(* Logix 5000 project; controller QW361 vendor 1 type 14 code 107 rev 32.11; software revision 32.00; part 9 of 20 *)

        [1052].log_data[0].time := 300.0, [1052].log_data[0].minminute := 10, [1052].log_data[0].maxminute := 10, [1052].log_data[0].valid := 1, [1052].log_data[1].valid := 1, [1052].log_data[2].valid := 1, [1052].log_data[3].valid := 1, [1052].log_data[4].valid := 1, [1052].time.Year := 2022, [1052].time.Month := 4, [1052].time.Day := 27, [1052].time.Hour := 13, [1052].time.Minute := 14, [1052].time.Second := 59, [1052].time.DST_ON := 1, [1053].log_data[0].min := 1.0, [1053].log_data[0].max := 1.0, [1053].log_data[0].total := 300.0, [1053].log_data[0].time := 300.0, [1053].log_data[0].minminute := 15, [1053].log_data[0].maxminute := 15, [1053].log_data[0].valid := 1, [1053].log_data[1].valid := 1, [1053].log_data[2].valid := 1, [1053].log_data[3].valid := 1, [1053].log_data[4].valid := 1, [1053].time.Year := 2022, [1053].time.Month := 4, [1053].time.Day := 27, [1053].time.Hour := 13, [1053].time.Minute := 19, [1053].time.Second := 59, [1053].time.DST_ON := 1, [1054].log_data[0].min := 1.0, [1054].log_data[0].max := 1.0, [1054].log_data[0].total := 300.0, [1054].log_data[0].time := 300.0, [1054].log_data[0].minminute := 20, [1054].log_data[0].maxminute := 20, [1054].log_data[0].valid := 1, [1054].log_data[1].valid := 1, [1054].log_data[2].valid := 1, [1054].log_data[3].valid := 1, [1054].log_data[4].valid := 1, [1054].time.Year := 2022, [1054].time.Month := 4, [1054].time.Day := 27, [1054].time.Hour := 13, [1054].time.Minute := 24, [1054].time.Second := 59, [1054].time.DST_ON := 1, [1055].log_data[0].min := 1.0, [1055].log_data[0].max := 1.0, [1055].log_data[0].total := 300.0, [1055].log_data[0].time := 300.0, [1055].log_data[0].minminute := 25, [1055].log_data[0].maxminute := 25, [1055].log_data[0].valid := 1, [1055].log_data[1].valid := 1, [1055].log_data[2].valid := 1,
        [1055].log_data[3].valid := 1, [1055].log_data[4].valid := 1, [1055].time.Year := 2022, [1055].time.Month := 4, [1055].time.Day := 27, [1055].time.Hour := 13, [1055].time.Minute := 29, [1055].time.Second := 59, [1055].time.DST_ON := 1, [1056].log_data[0].min := 1.0, [1056].log_data[0].max := 1.0, [1056].log_data[0].total := 300.0, [1056].log_data[0].time := 300.0, [1056].log_data[0].minminute := 30, [1056].log_data[0].maxminute := 30, [1056].log_data[0].valid := 1, [1056].log_data[1].valid := 1, [1056].log_data[2].valid := 1, [1056].log_data[3].valid := 1, [1056].log_data[4].valid := 1, [1056].time.Year := 2022, [1056].time.Month := 4, [1056].time.Day := 27, [1056].time.Hour := 13, [1056].time.Minute := 34, [1056].time.Second := 59, [1056].time.DST_ON := 1, [1057].log_data[0].min := 1.0, [1057].log_data[0].max := 1.0, [1057].log_data[0].total := 300.0, [1057].log_data[0].time := 300.0, [1057].log_data[0].minminute := 35, [1057].log_data[0].maxminute := 35, [1057].log_data[0].valid := 1, [1057].log_data[1].valid := 1, [1057].log_data[2].valid := 1, [1057].log_data[3].valid := 1, [1057].log_data[4].valid := 1, [1057].time.Year := 2022, [1057].time.Month := 4, [1057].time.Day := 27, [1057].time.Hour := 13, [1057].time.Minute := 39, [1057].time.Second := 59, [1057].time.DST_ON := 1, [1058].log_data[0].min := 1.0, [1058].log_data[0].max := 1.0, [1058].log_data[0].total := 300.0, [1058].log_data[0].time := 300.0, [1058].log_data[0].minminute := 40, [1058].log_data[0].maxminute := 40, [1058].log_data[0].valid := 1, [1058].log_data[1].valid := 1, [1058].log_data[2].valid := 1, [1058].log_data[3].valid := 1, [1058].log_data[4].valid := 1, [1058].time.Year := 2022, [1058].time.Month := 4, [1058].time.Day := 27, [1058].time.Hour := 13,
        [1058].time.Minute := 44, [1058].time.Second := 59, [1058].time.DST_ON := 1, [1059].log_data[0].min := 1.0, [1059].log_data[0].max := 1.0, [1059].log_data[0].total := 300.0, [1059].log_data[0].time := 300.0, [1059].log_data[0].minminute := 45, [1059].log_data[0].maxminute := 45, [1059].log_data[0].valid := 1, [1059].log_data[1].valid := 1, [1059].log_data[2].valid := 1, [1059].log_data[3].valid := 1, [1059].log_data[4].valid := 1, [1059].time.Year := 2022, [1059].time.Month := 4, [1059].time.Day := 27, [1059].time.Hour := 13, [1059].time.Minute := 49, [1059].time.Second := 59, [1059].time.DST_ON := 1, [1060].log_data[0].min := 1.0, [1060].log_data[0].max := 1.0, [1060].log_data[0].total := 300.0, [1060].log_data[0].time := 300.0, [1060].log_data[0].minminute := 50, [1060].log_data[0].maxminute := 50, [1060].log_data[0].valid := 1, [1060].log_data[1].valid := 1, [1060].log_data[2].valid := 1, [1060].log_data[3].valid := 1, [1060].log_data[4].valid := 1, [1060].time.Year := 2022, [1060].time.Month := 4, [1060].time.Day := 27, [1060].time.Hour := 13, [1060].time.Minute := 54, [1060].time.Second := 59, [1060].time.DST_ON := 1, [1061].log_data[0].min := 1.0, [1061].log_data[0].max := 1.0, [1061].log_data[0].total := 300.0, [1061].log_data[0].time := 300.0, [1061].log_data[0].minminute := 55, [1061].log_data[0].maxminute := 55, [1061].log_data[0].valid := 1, [1061].log_data[1].valid := 1, [1061].log_data[2].valid := 1, [1061].log_data[3].valid := 1, [1061].log_data[4].valid := 1, [1061].time.Year := 2022, [1061].time.Month := 4, [1061].time.Day := 27, [1061].time.Hour := 13, [1061].time.Minute := 59, [1061].time.Second := 59, [1061].time.DST_ON := 1, [1062].log_data[0].min := 1.0, [1062].log_data[0].max := 1.0, [1062].log_data[0].total := 300.0,
        [1062].log_data[0].time := 300.0, [1062].log_data[0].valid := 1, [1062].log_data[1].valid := 1, [1062].log_data[2].valid := 1, [1062].log_data[3].valid := 1, [1062].log_data[4].valid := 1, [1062].time.Year := 2022, [1062].time.Month := 4, [1062].time.Day := 27, [1062].time.Hour := 14, [1062].time.Minute := 4, [1062].time.Second := 59, [1062].time.DST_ON := 1, [1063].log_data[0].min := 1.0, [1063].log_data[0].max := 1.0, [1063].log_data[0].total := 300.0, [1063].log_data[0].time := 300.0, [1063].log_data[0].minminute := 5, [1063].log_data[0].maxminute := 5, [1063].log_data[0].valid := 1, [1063].log_data[1].valid := 1, [1063].log_data[2].valid := 1, [1063].log_data[3].valid := 1, [1063].log_data[4].valid := 1, [1063].time.Year := 2022, [1063].time.Month := 4, [1063].time.Day := 27, [1063].time.Hour := 14, [1063].time.Minute := 9, [1063].time.Second := 59, [1063].time.DST_ON := 1, [1064].log_data[0].min := 1.0, [1064].log_data[0].max := 1.0, [1064].log_data[0].total := 300.0, [1064].log_data[0].time := 300.0, [1064].log_data[0].minminute := 10, [1064].log_data[0].maxminute := 10, [1064].log_data[0].valid := 1, [1064].log_data[1].valid := 1, [1064].log_data[2].valid := 1, [1064].log_data[3].valid := 1, [1064].log_data[4].valid := 1, [1064].time.Year := 2022, [1064].time.Month := 4, [1064].time.Day := 27, [1064].time.Hour := 14, [1064].time.Minute := 14, [1064].time.Second := 59, [1064].time.DST_ON := 1, [1065].log_data[0].min := 1.0, [1065].log_data[0].max := 1.0, [1065].log_data[0].total := 300.0, [1065].log_data[0].time := 300.0, [1065].log_data[0].minminute := 15, [1065].log_data[0].maxminute := 15, [1065].log_data[0].valid := 1, [1065].log_data[1].valid := 1, [1065].log_data[2].valid := 1, [1065].log_data[3].valid := 1, [1065].log_data[4].valid := 1,
        [1065].time.Year := 2022, [1065].time.Month := 4, [1065].time.Day := 27, [1065].time.Hour := 14, [1065].time.Minute := 19, [1065].time.Second := 59, [1065].time.DST_ON := 1, [1066].log_data[0].min := 1.0, [1066].log_data[0].max := 1.0, [1066].log_data[0].total := 300.0, [1066].log_data[0].time := 300.0, [1066].log_data[0].minminute := 20, [1066].log_data[0].maxminute := 20, [1066].log_data[0].valid := 1, [1066].log_data[1].valid := 1, [1066].log_data[2].valid := 1, [1066].log_data[3].valid := 1, [1066].log_data[4].valid := 1, [1066].time.Year := 2022, [1066].time.Month := 4, [1066].time.Day := 27, [1066].time.Hour := 14, [1066].time.Minute := 24, [1066].time.Second := 59, [1066].time.DST_ON := 1, [1067].log_data[0].min := 1.0, [1067].log_data[0].max := 1.0, [1067].log_data[0].total := 300.0, [1067].log_data[0].time := 300.0, [1067].log_data[0].minminute := 25, [1067].log_data[0].maxminute := 25, [1067].log_data[0].valid := 1, [1067].log_data[1].valid := 1, [1067].log_data[2].valid := 1, [1067].log_data[3].valid := 1, [1067].log_data[4].valid := 1, [1067].time.Year := 2022, [1067].time.Month := 4, [1067].time.Day := 27, [1067].time.Hour := 14, [1067].time.Minute := 29, [1067].time.Second := 59, [1067].time.DST_ON := 1, [1068].log_data[0].min := 1.0, [1068].log_data[0].max := 1.0, [1068].log_data[0].total := 300.0, [1068].log_data[0].time := 300.0, [1068].log_data[0].minminute := 30, [1068].log_data[0].maxminute := 30, [1068].log_data[0].valid := 1, [1068].log_data[1].valid := 1, [1068].log_data[2].valid := 1, [1068].log_data[3].valid := 1, [1068].log_data[4].valid := 1, [1068].time.Year := 2022, [1068].time.Month := 4, [1068].time.Day := 27, [1068].time.Hour := 14, [1068].time.Minute := 34, [1068].time.Second := 59,
        [1068].time.DST_ON := 1, [1069].log_data[0].min := 1.0, [1069].log_data[0].max := 1.0, [1069].log_data[0].total := 300.0, [1069].log_data[0].time := 300.0, [1069].log_data[0].minminute := 35, [1069].log_data[0].maxminute := 35, [1069].log_data[0].valid := 1, [1069].log_data[1].valid := 1, [1069].log_data[2].valid := 1, [1069].log_data[3].valid := 1, [1069].log_data[4].valid := 1, [1069].time.Year := 2022, [1069].time.Month := 4, [1069].time.Day := 27, [1069].time.Hour := 14, [1069].time.Minute := 39, [1069].time.Second := 59, [1069].time.DST_ON := 1, [1070].log_data[0].min := 1.0, [1070].log_data[0].max := 1.0, [1070].log_data[0].total := 300.0, [1070].log_data[0].time := 300.0, [1070].log_data[0].minminute := 40, [1070].log_data[0].maxminute := 40, [1070].log_data[0].valid := 1, [1070].log_data[1].valid := 1, [1070].log_data[2].valid := 1, [1070].log_data[3].valid := 1, [1070].log_data[4].valid := 1, [1070].time.Year := 2022, [1070].time.Month := 4, [1070].time.Day := 27, [1070].time.Hour := 14, [1070].time.Minute := 44, [1070].time.Second := 59, [1070].time.DST_ON := 1, [1071].log_data[0].min := 1.0, [1071].log_data[0].max := 1.0, [1071].log_data[0].total := 300.0, [1071].log_data[0].time := 300.0, [1071].log_data[0].minminute := 45, [1071].log_data[0].maxminute := 45, [1071].log_data[0].valid := 1, [1071].log_data[1].valid := 1, [1071].log_data[2].valid := 1, [1071].log_data[3].valid := 1, [1071].log_data[4].valid := 1, [1071].time.Year := 2022, [1071].time.Month := 4, [1071].time.Day := 27, [1071].time.Hour := 14, [1071].time.Minute := 49, [1071].time.Second := 59, [1071].time.DST_ON := 1, [1072].log_data[0].min := 1.0, [1072].log_data[0].max := 1.0, [1072].log_data[0].total := 300.0, [1072].log_data[0].time := 300.0, [1072].log_data[0].minminute := 50,
        [1072].log_data[0].maxminute := 50, [1072].log_data[0].valid := 1, [1072].log_data[1].valid := 1, [1072].log_data[2].valid := 1, [1072].log_data[3].valid := 1, [1072].log_data[4].valid := 1, [1072].time.Year := 2022, [1072].time.Month := 4, [1072].time.Day := 27, [1072].time.Hour := 14, [1072].time.Minute := 54, [1072].time.Second := 59, [1072].time.DST_ON := 1, [1073].log_data[0].min := 1.0, [1073].log_data[0].max := 1.0, [1073].log_data[0].total := 300.0, [1073].log_data[0].time := 300.0, [1073].log_data[0].minminute := 55, [1073].log_data[0].maxminute := 55, [1073].log_data[0].valid := 1, [1073].log_data[1].valid := 1, [1073].log_data[2].valid := 1, [1073].log_data[3].valid := 1, [1073].log_data[4].valid := 1, [1073].time.Year := 2022, [1073].time.Month := 4, [1073].time.Day := 27, [1073].time.Hour := 14, [1073].time.Minute := 59, [1073].time.Second := 59, [1073].time.DST_ON := 1, [1074].log_data[0].min := 1.0, [1074].log_data[0].max := 1.0, [1074].log_data[0].total := 300.0, [1074].log_data[0].time := 300.0, [1074].log_data[0].valid := 1, [1074].log_data[1].valid := 1, [1074].log_data[2].valid := 1, [1074].log_data[3].valid := 1, [1074].log_data[4].valid := 1, [1074].time.Year := 2022, [1074].time.Month := 4, [1074].time.Day := 27, [1074].time.Hour := 15, [1074].time.Minute := 4, [1074].time.Second := 59, [1074].time.DST_ON := 1, [1075].log_data[0].min := 1.0, [1075].log_data[0].max := 1.0, [1075].log_data[0].total := 300.0, [1075].log_data[0].time := 300.0, [1075].log_data[0].minminute := 5, [1075].log_data[0].maxminute := 5, [1075].log_data[0].valid := 1, [1075].log_data[1].valid := 1, [1075].log_data[2].valid := 1, [1075].log_data[3].valid := 1, [1075].log_data[4].valid := 1, [1075].time.Year := 2022, [1075].time.Month := 4,
        [1075].time.Day := 27, [1075].time.Hour := 15, [1075].time.Minute := 9, [1075].time.Second := 59, [1075].time.DST_ON := 1, [1076].log_data[0].min := 1.0, [1076].log_data[0].max := 1.0, [1076].log_data[0].total := 300.0, [1076].log_data[0].time := 300.0, [1076].log_data[0].minminute := 10, [1076].log_data[0].maxminute := 10, [1076].log_data[0].valid := 1, [1076].log_data[1].valid := 1, [1076].log_data[2].valid := 1, [1076].log_data[3].valid := 1, [1076].log_data[4].valid := 1, [1076].time.Year := 2022, [1076].time.Month := 4, [1076].time.Day := 27, [1076].time.Hour := 15, [1076].time.Minute := 14, [1076].time.Second := 59, [1076].time.DST_ON := 1, [1077].log_data[0].min := 1.0, [1077].log_data[0].max := 1.0, [1077].log_data[0].total := 300.0, [1077].log_data[0].time := 300.0, [1077].log_data[0].minminute := 15, [1077].log_data[0].maxminute := 15, [1077].log_data[0].valid := 1, [1077].log_data[1].valid := 1, [1077].log_data[2].valid := 1, [1077].log_data[3].valid := 1, [1077].log_data[4].valid := 1, [1077].time.Year := 2022, [1077].time.Month := 4, [1077].time.Day := 27, [1077].time.Hour := 15, [1077].time.Minute := 19, [1077].time.Second := 59, [1077].time.DST_ON := 1, [1078].log_data[0].min := 1.0, [1078].log_data[0].max := 1.0, [1078].log_data[0].total := 300.0, [1078].log_data[0].time := 300.0, [1078].log_data[0].minminute := 20, [1078].log_data[0].maxminute := 20, [1078].log_data[0].valid := 1, [1078].log_data[1].valid := 1, [1078].log_data[2].valid := 1, [1078].log_data[3].valid := 1, [1078].log_data[4].valid := 1, [1078].time.Year := 2022, [1078].time.Month := 4, [1078].time.Day := 27, [1078].time.Hour := 15, [1078].time.Minute := 24, [1078].time.Second := 59, [1078].time.DST_ON := 1, [1079].log_data[0].min := 1.0,
        [1079].log_data[0].max := 1.0, [1079].log_data[0].total := 300.0, [1079].log_data[0].time := 300.0, [1079].log_data[0].minminute := 25, [1079].log_data[0].maxminute := 25, [1079].log_data[0].valid := 1, [1079].log_data[1].valid := 1, [1079].log_data[2].valid := 1, [1079].log_data[3].valid := 1, [1079].log_data[4].valid := 1, [1079].time.Year := 2022, [1079].time.Month := 4, [1079].time.Day := 27, [1079].time.Hour := 15, [1079].time.Minute := 29, [1079].time.Second := 59, [1079].time.DST_ON := 1, [1080].log_data[0].min := 1.0, [1080].log_data[0].max := 1.0, [1080].log_data[0].total := 299.999, [1080].log_data[0].time := 299.999, [1080].log_data[0].minminute := 30, [1080].log_data[0].maxminute := 30, [1080].log_data[0].valid := 1, [1080].log_data[1].valid := 1, [1080].log_data[2].valid := 1, [1080].log_data[3].valid := 1, [1080].log_data[4].valid := 1, [1080].time.Year := 2022, [1080].time.Month := 4, [1080].time.Day := 27, [1080].time.Hour := 15, [1080].time.Minute := 34, [1080].time.Second := 59, [1080].time.DST_ON := 1, [1081].log_data[0].min := 1.0, [1081].log_data[0].max := 1.0, [1081].log_data[0].total := 300.0, [1081].log_data[0].time := 300.0, [1081].log_data[0].minminute := 35, [1081].log_data[0].maxminute := 35, [1081].log_data[0].valid := 1, [1081].log_data[1].valid := 1, [1081].log_data[2].valid := 1, [1081].log_data[3].valid := 1, [1081].log_data[4].valid := 1, [1081].time.Year := 2022, [1081].time.Month := 4, [1081].time.Day := 27, [1081].time.Hour := 15, [1081].time.Minute := 39, [1081].time.Second := 59, [1081].time.DST_ON := 1, [1082].log_data[0].min := 1.0, [1082].log_data[0].max := 1.0, [1082].log_data[0].total := 300.0, [1082].log_data[0].time := 300.0, [1082].log_data[0].minminute := 40, [1082].log_data[0].maxminute := 40, [1082].log_data[0].valid := 1,
        [1082].log_data[1].valid := 1, [1082].log_data[2].valid := 1, [1082].log_data[3].valid := 1, [1082].log_data[4].valid := 1, [1082].time.Year := 2022, [1082].time.Month := 4, [1082].time.Day := 27, [1082].time.Hour := 15, [1082].time.Minute := 44, [1082].time.Second := 59, [1082].time.DST_ON := 1, [1083].log_data[0].min := 1.0, [1083].log_data[0].max := 1.0, [1083].log_data[0].total := 300.0, [1083].log_data[0].time := 300.0, [1083].log_data[0].minminute := 45, [1083].log_data[0].maxminute := 45, [1083].log_data[0].valid := 1, [1083].log_data[1].valid := 1, [1083].log_data[2].valid := 1, [1083].log_data[3].valid := 1, [1083].log_data[4].valid := 1, [1083].time.Year := 2022, [1083].time.Month := 4, [1083].time.Day := 27, [1083].time.Hour := 15, [1083].time.Minute := 49, [1083].time.Second := 59, [1083].time.DST_ON := 1, [1084].log_data[0].min := 1.0, [1084].log_data[0].max := 1.0, [1084].log_data[0].total := 300.0, [1084].log_data[0].time := 300.0, [1084].log_data[0].minminute := 50, [1084].log_data[0].maxminute := 50, [1084].log_data[0].valid := 1, [1084].log_data[1].valid := 1, [1084].log_data[2].valid := 1, [1084].log_data[3].valid := 1, [1084].log_data[4].valid := 1, [1084].time.Year := 2022, [1084].time.Month := 4, [1084].time.Day := 27, [1084].time.Hour := 15, [1084].time.Minute := 54, [1084].time.Second := 59, [1084].time.DST_ON := 1, [1085].log_data[0].min := 1.0, [1085].log_data[0].max := 1.0, [1085].log_data[0].total := 300.0, [1085].log_data[0].time := 300.0, [1085].log_data[0].minminute := 55, [1085].log_data[0].maxminute := 55, [1085].log_data[0].valid := 1, [1085].log_data[1].valid := 1, [1085].log_data[2].valid := 1, [1085].log_data[3].valid := 1, [1085].log_data[4].valid := 1, [1085].time.Year := 2022, [1085].time.Month := 4,
        [1085].time.Day := 27, [1085].time.Hour := 15, [1085].time.Minute := 59, [1085].time.Second := 59, [1085].time.DST_ON := 1, [1086].log_data[0].min := 1.0, [1086].log_data[0].max := 1.0, [1086].log_data[0].total := 300.0, [1086].log_data[0].time := 300.0, [1086].log_data[0].valid := 1, [1086].log_data[1].valid := 1, [1086].log_data[2].valid := 1, [1086].log_data[3].valid := 1, [1086].log_data[4].valid := 1, [1086].time.Year := 2022, [1086].time.Month := 4, [1086].time.Day := 27, [1086].time.Hour := 16, [1086].time.Minute := 4, [1086].time.Second := 59, [1086].time.DST_ON := 1, [1087].log_data[0].min := 1.0, [1087].log_data[0].max := 1.0, [1087].log_data[0].total := 300.0, [1087].log_data[0].time := 300.0, [1087].log_data[0].minminute := 5, [1087].log_data[0].maxminute := 5, [1087].log_data[0].valid := 1, [1087].log_data[1].valid := 1, [1087].log_data[2].valid := 1, [1087].log_data[3].valid := 1, [1087].log_data[4].valid := 1, [1087].time.Year := 2022, [1087].time.Month := 4, [1087].time.Day := 27, [1087].time.Hour := 16, [1087].time.Minute := 9, [1087].time.Second := 59, [1087].time.DST_ON := 1, [1088].log_data[0].min := 1.0, [1088].log_data[0].max := 1.0, [1088].log_data[0].total := 300.0, [1088].log_data[0].time := 300.0, [1088].log_data[0].minminute := 10, [1088].log_data[0].maxminute := 10, [1088].log_data[0].valid := 1, [1088].log_data[1].valid := 1, [1088].log_data[2].valid := 1, [1088].log_data[3].valid := 1, [1088].log_data[4].valid := 1, [1088].time.Year := 2022, [1088].time.Month := 4, [1088].time.Day := 27, [1088].time.Hour := 16, [1088].time.Minute := 14, [1088].time.Second := 59, [1088].time.DST_ON := 1, [1089].log_data[0].min := 1.0, [1089].log_data[0].max := 1.0, [1089].log_data[0].total := 300.0,
        [1089].log_data[0].time := 300.0, [1089].log_data[0].minminute := 15, [1089].log_data[0].maxminute := 15, [1089].log_data[0].valid := 1, [1089].log_data[1].valid := 1, [1089].log_data[2].valid := 1, [1089].log_data[3].valid := 1, [1089].log_data[4].valid := 1, [1089].time.Year := 2022, [1089].time.Month := 4, [1089].time.Day := 27, [1089].time.Hour := 16, [1089].time.Minute := 19, [1089].time.Second := 59, [1089].time.DST_ON := 1, [1090].log_data[0].min := 1.0, [1090].log_data[0].max := 1.0, [1090].log_data[0].total := 300.0, [1090].log_data[0].time := 300.0, [1090].log_data[0].minminute := 20, [1090].log_data[0].maxminute := 20, [1090].log_data[0].valid := 1, [1090].log_data[1].valid := 1, [1090].log_data[2].valid := 1, [1090].log_data[3].valid := 1, [1090].log_data[4].valid := 1, [1090].time.Year := 2022, [1090].time.Month := 4, [1090].time.Day := 27, [1090].time.Hour := 16, [1090].time.Minute := 24, [1090].time.Second := 59, [1090].time.DST_ON := 1, [1091].log_data[0].min := 1.0, [1091].log_data[0].max := 1.0, [1091].log_data[0].total := 300.0, [1091].log_data[0].time := 300.0, [1091].log_data[0].minminute := 25, [1091].log_data[0].maxminute := 25, [1091].log_data[0].valid := 1, [1091].log_data[1].valid := 1, [1091].log_data[2].valid := 1, [1091].log_data[3].valid := 1, [1091].log_data[4].valid := 1, [1091].time.Year := 2022, [1091].time.Month := 4, [1091].time.Day := 27, [1091].time.Hour := 16, [1091].time.Minute := 29, [1091].time.Second := 59, [1091].time.DST_ON := 1, [1092].log_data[0].min := 1.0, [1092].log_data[0].max := 1.0, [1092].log_data[0].total := 300.0, [1092].log_data[0].time := 300.0, [1092].log_data[0].minminute := 30, [1092].log_data[0].maxminute := 30, [1092].log_data[0].valid := 1, [1092].log_data[1].valid := 1, [1092].log_data[2].valid := 1,
        [1092].log_data[3].valid := 1, [1092].log_data[4].valid := 1, [1092].time.Year := 2022, [1092].time.Month := 4, [1092].time.Day := 27, [1092].time.Hour := 16, [1092].time.Minute := 34, [1092].time.Second := 59, [1092].time.DST_ON := 1, [1093].log_data[0].min := 1.0, [1093].log_data[0].max := 1.0, [1093].log_data[0].total := 300.0, [1093].log_data[0].time := 300.0, [1093].log_data[0].minminute := 35, [1093].log_data[0].maxminute := 35, [1093].log_data[0].valid := 1, [1093].log_data[1].valid := 1, [1093].log_data[2].valid := 1, [1093].log_data[3].valid := 1, [1093].log_data[4].valid := 1, [1093].time.Year := 2022, [1093].time.Month := 4, [1093].time.Day := 27, [1093].time.Hour := 16, [1093].time.Minute := 39, [1093].time.Second := 59, [1093].time.DST_ON := 1, [1094].log_data[0].min := 1.0, [1094].log_data[0].max := 1.0, [1094].log_data[0].total := 300.0, [1094].log_data[0].time := 300.0, [1094].log_data[0].minminute := 40, [1094].log_data[0].maxminute := 40, [1094].log_data[0].valid := 1, [1094].log_data[1].valid := 1, [1094].log_data[2].valid := 1, [1094].log_data[3].valid := 1, [1094].log_data[4].valid := 1, [1094].time.Year := 2022, [1094].time.Month := 4, [1094].time.Day := 27, [1094].time.Hour := 16, [1094].time.Minute := 44, [1094].time.Second := 59, [1094].time.DST_ON := 1, [1095].log_data[0].min := 1.0, [1095].log_data[0].max := 1.0, [1095].log_data[0].total := 300.0, [1095].log_data[0].time := 300.0, [1095].log_data[0].minminute := 45, [1095].log_data[0].maxminute := 45, [1095].log_data[0].valid := 1, [1095].log_data[1].valid := 1, [1095].log_data[2].valid := 1, [1095].log_data[3].valid := 1, [1095].log_data[4].valid := 1, [1095].time.Year := 2022, [1095].time.Month := 4, [1095].time.Day := 27, [1095].time.Hour := 16,
        [1095].time.Minute := 49, [1095].time.Second := 59, [1095].time.DST_ON := 1, [1096].log_data[0].min := 1.0, [1096].log_data[0].max := 1.0, [1096].log_data[0].total := 300.0, [1096].log_data[0].time := 300.0, [1096].log_data[0].minminute := 50, [1096].log_data[0].maxminute := 50, [1096].log_data[0].valid := 1, [1096].log_data[1].valid := 1, [1096].log_data[2].valid := 1, [1096].log_data[3].valid := 1, [1096].log_data[4].valid := 1, [1096].time.Year := 2022, [1096].time.Month := 4, [1096].time.Day := 27, [1096].time.Hour := 16, [1096].time.Minute := 54, [1096].time.Second := 59, [1096].time.DST_ON := 1, [1097].log_data[0].min := 1.0, [1097].log_data[0].max := 1.0, [1097].log_data[0].total := 300.0, [1097].log_data[0].time := 300.0, [1097].log_data[0].minminute := 55, [1097].log_data[0].maxminute := 55, [1097].log_data[0].valid := 1, [1097].log_data[1].valid := 1, [1097].log_data[2].valid := 1, [1097].log_data[3].valid := 1, [1097].log_data[4].valid := 1, [1097].time.Year := 2022, [1097].time.Month := 4, [1097].time.Day := 27, [1097].time.Hour := 16, [1097].time.Minute := 59, [1097].time.Second := 59, [1097].time.DST_ON := 1, [1098].log_data[0].min := 1.0, [1098].log_data[0].max := 1.0, [1098].log_data[0].total := 300.0, [1098].log_data[0].time := 300.0, [1098].log_data[0].valid := 1, [1098].log_data[1].valid := 1, [1098].log_data[2].valid := 1, [1098].log_data[3].valid := 1, [1098].log_data[4].valid := 1, [1098].time.Year := 2022, [1098].time.Month := 4, [1098].time.Day := 27, [1098].time.Hour := 17, [1098].time.Minute := 4, [1098].time.Second := 59, [1098].time.DST_ON := 1, [1099].log_data[0].min := 1.0, [1099].log_data[0].max := 1.0, [1099].log_data[0].total := 300.0, [1099].log_data[0].time := 300.0, [1099].log_data[0].minminute := 5,
        [1099].log_data[0].maxminute := 5, [1099].log_data[0].valid := 1, [1099].log_data[1].valid := 1, [1099].log_data[2].valid := 1, [1099].log_data[3].valid := 1, [1099].log_data[4].valid := 1, [1099].time.Year := 2022, [1099].time.Month := 4, [1099].time.Day := 27, [1099].time.Hour := 17, [1099].time.Minute := 9, [1099].time.Second := 59, [1099].time.DST_ON := 1, [1100].log_data[0].min := 1.0, [1100].log_data[0].max := 1.0, [1100].log_data[0].total := 300.0, [1100].log_data[0].time := 300.0, [1100].log_data[0].minminute := 10, [1100].log_data[0].maxminute := 10, [1100].log_data[0].valid := 1, [1100].log_data[1].valid := 1, [1100].log_data[2].valid := 1, [1100].log_data[3].valid := 1, [1100].log_data[4].valid := 1, [1100].time.Year := 2022, [1100].time.Month := 4, [1100].time.Day := 27, [1100].time.Hour := 17, [1100].time.Minute := 14, [1100].time.Second := 59, [1100].time.DST_ON := 1, [1101].log_data[0].min := 1.0, [1101].log_data[0].max := 1.0, [1101].log_data[0].total := 300.0, [1101].log_data[0].time := 300.0, [1101].log_data[0].minminute := 15, [1101].log_data[0].maxminute := 15, [1101].log_data[0].valid := 1, [1101].log_data[1].valid := 1, [1101].log_data[2].valid := 1, [1101].log_data[3].valid := 1, [1101].log_data[4].valid := 1, [1101].time.Year := 2022, [1101].time.Month := 4, [1101].time.Day := 27, [1101].time.Hour := 17, [1101].time.Minute := 19, [1101].time.Second := 59, [1101].time.DST_ON := 1, [1102].log_data[0].min := 1.0, [1102].log_data[0].max := 1.0, [1102].log_data[0].total := 300.0, [1102].log_data[0].time := 300.0, [1102].log_data[0].minminute := 20, [1102].log_data[0].maxminute := 20, [1102].log_data[0].valid := 1, [1102].log_data[1].valid := 1, [1102].log_data[2].valid := 1, [1102].log_data[3].valid := 1, [1102].log_data[4].valid := 1,
        [1102].time.Year := 2022, [1102].time.Month := 4, [1102].time.Day := 27, [1102].time.Hour := 17, [1102].time.Minute := 24, [1102].time.Second := 59, [1102].time.DST_ON := 1, [1103].log_data[0].min := 1.0, [1103].log_data[0].max := 1.0, [1103].log_data[0].total := 300.0, [1103].log_data[0].time := 300.0, [1103].log_data[0].minminute := 25, [1103].log_data[0].maxminute := 25, [1103].log_data[0].valid := 1, [1103].log_data[1].valid := 1, [1103].log_data[2].valid := 1, [1103].log_data[3].valid := 1, [1103].log_data[4].valid := 1, [1103].time.Year := 2022, [1103].time.Month := 4, [1103].time.Day := 27, [1103].time.Hour := 17, [1103].time.Minute := 29, [1103].time.Second := 59, [1103].time.DST_ON := 1, [1104].log_data[0].min := 1.0, [1104].log_data[0].max := 1.0, [1104].log_data[0].total := 300.0, [1104].log_data[0].time := 300.0, [1104].log_data[0].minminute := 30, [1104].log_data[0].maxminute := 30, [1104].log_data[0].valid := 1, [1104].log_data[1].valid := 1, [1104].log_data[2].valid := 1, [1104].log_data[3].valid := 1, [1104].log_data[4].valid := 1, [1104].time.Year := 2022, [1104].time.Month := 4, [1104].time.Day := 27, [1104].time.Hour := 17, [1104].time.Minute := 34, [1104].time.Second := 59, [1104].time.DST_ON := 1, [1105].log_data[0].min := 1.0, [1105].log_data[0].max := 1.0, [1105].log_data[0].total := 300.0, [1105].log_data[0].time := 300.0, [1105].log_data[0].minminute := 35, [1105].log_data[0].maxminute := 35, [1105].log_data[0].valid := 1, [1105].log_data[1].valid := 1, [1105].log_data[2].valid := 1, [1105].log_data[3].valid := 1, [1105].log_data[4].valid := 1, [1105].time.Year := 2022, [1105].time.Month := 4, [1105].time.Day := 27, [1105].time.Hour := 17, [1105].time.Minute := 39, [1105].time.Second := 59,
        [1105].time.DST_ON := 1, [1106].log_data[0].min := 1.0, [1106].log_data[0].max := 1.0, [1106].log_data[0].total := 299.999, [1106].log_data[0].time := 299.999, [1106].log_data[0].minminute := 40, [1106].log_data[0].maxminute := 40, [1106].log_data[0].valid := 1, [1106].log_data[1].valid := 1, [1106].log_data[2].valid := 1, [1106].log_data[3].valid := 1, [1106].log_data[4].valid := 1, [1106].time.Year := 2022, [1106].time.Month := 4, [1106].time.Day := 27, [1106].time.Hour := 17, [1106].time.Minute := 44, [1106].time.Second := 59, [1106].time.DST_ON := 1, [1107].log_data[0].min := 1.0, [1107].log_data[0].max := 1.0, [1107].log_data[0].total := 300.0, [1107].log_data[0].time := 300.0, [1107].log_data[0].minminute := 45, [1107].log_data[0].maxminute := 45, [1107].log_data[0].valid := 1, [1107].log_data[1].valid := 1, [1107].log_data[2].valid := 1, [1107].log_data[3].valid := 1, [1107].log_data[4].valid := 1, [1107].time.Year := 2022, [1107].time.Month := 4, [1107].time.Day := 27, [1107].time.Hour := 17, [1107].time.Minute := 49, [1107].time.Second := 59, [1107].time.DST_ON := 1, [1108].log_data[0].min := 1.0, [1108].log_data[0].max := 1.0, [1108].log_data[0].total := 300.0, [1108].log_data[0].time := 300.0, [1108].log_data[0].minminute := 50, [1108].log_data[0].maxminute := 50, [1108].log_data[0].valid := 1, [1108].log_data[1].valid := 1, [1108].log_data[2].valid := 1, [1108].log_data[3].valid := 1, [1108].log_data[4].valid := 1, [1108].time.Year := 2022, [1108].time.Month := 4, [1108].time.Day := 27, [1108].time.Hour := 17, [1108].time.Minute := 54, [1108].time.Second := 59, [1108].time.DST_ON := 1, [1109].log_data[0].min := 1.0, [1109].log_data[0].max := 1.0, [1109].log_data[0].total := 300.0, [1109].log_data[0].time := 300.0, [1109].log_data[0].minminute := 55,
        [1109].log_data[0].maxminute := 55, [1109].log_data[0].valid := 1, [1109].log_data[1].valid := 1, [1109].log_data[2].valid := 1, [1109].log_data[3].valid := 1, [1109].log_data[4].valid := 1, [1109].time.Year := 2022, [1109].time.Month := 4, [1109].time.Day := 27, [1109].time.Hour := 17, [1109].time.Minute := 59, [1109].time.Second := 59, [1109].time.DST_ON := 1, [1110].log_data[0].min := 1.0, [1110].log_data[0].max := 1.0, [1110].log_data[0].total := 300.0, [1110].log_data[0].time := 300.0, [1110].log_data[0].valid := 1, [1110].log_data[1].valid := 1, [1110].log_data[2].valid := 1, [1110].log_data[3].valid := 1, [1110].log_data[4].valid := 1, [1110].time.Year := 2022, [1110].time.Month := 4, [1110].time.Day := 27, [1110].time.Hour := 18, [1110].time.Minute := 4, [1110].time.Second := 59, [1110].time.DST_ON := 1, [1111].log_data[0].min := 1.0, [1111].log_data[0].max := 1.0, [1111].log_data[0].total := 300.0, [1111].log_data[0].time := 300.0, [1111].log_data[0].minminute := 5, [1111].log_data[0].maxminute := 5, [1111].log_data[0].valid := 1, [1111].log_data[1].valid := 1, [1111].log_data[2].valid := 1, [1111].log_data[3].valid := 1, [1111].log_data[4].valid := 1, [1111].time.Year := 2022, [1111].time.Month := 4, [1111].time.Day := 27, [1111].time.Hour := 18, [1111].time.Minute := 9, [1111].time.Second := 59, [1111].time.DST_ON := 1, [1112].log_data[0].min := 1.0, [1112].log_data[0].max := 1.0, [1112].log_data[0].total := 300.0, [1112].log_data[0].time := 300.0, [1112].log_data[0].minminute := 10, [1112].log_data[0].maxminute := 10, [1112].log_data[0].valid := 1, [1112].log_data[1].valid := 1, [1112].log_data[2].valid := 1, [1112].log_data[3].valid := 1, [1112].log_data[4].valid := 1, [1112].time.Year := 2022, [1112].time.Month := 4,
        [1112].time.Day := 27, [1112].time.Hour := 18, [1112].time.Minute := 14, [1112].time.Second := 59, [1112].time.DST_ON := 1, [1113].log_data[0].min := 1.0, [1113].log_data[0].max := 1.0, [1113].log_data[0].total := 300.0, [1113].log_data[0].time := 300.0, [1113].log_data[0].minminute := 15, [1113].log_data[0].maxminute := 15, [1113].log_data[0].valid := 1, [1113].log_data[1].valid := 1, [1113].log_data[2].valid := 1, [1113].log_data[3].valid := 1, [1113].log_data[4].valid := 1, [1113].time.Year := 2022, [1113].time.Month := 4, [1113].time.Day := 27, [1113].time.Hour := 18, [1113].time.Minute := 19, [1113].time.Second := 59, [1113].time.DST_ON := 1, [1114].log_data[0].min := 1.0, [1114].log_data[0].max := 1.0, [1114].log_data[0].total := 300.0, [1114].log_data[0].time := 300.0, [1114].log_data[0].minminute := 20, [1114].log_data[0].maxminute := 20, [1114].log_data[0].valid := 1, [1114].log_data[1].valid := 1, [1114].log_data[2].valid := 1, [1114].log_data[3].valid := 1, [1114].log_data[4].valid := 1, [1114].time.Year := 2022, [1114].time.Month := 4, [1114].time.Day := 27, [1114].time.Hour := 18, [1114].time.Minute := 24, [1114].time.Second := 59, [1114].time.DST_ON := 1, [1115].log_data[0].min := 1.0, [1115].log_data[0].max := 1.0, [1115].log_data[0].total := 300.0, [1115].log_data[0].time := 300.0, [1115].log_data[0].minminute := 25, [1115].log_data[0].maxminute := 25, [1115].log_data[0].valid := 1, [1115].log_data[1].valid := 1, [1115].log_data[2].valid := 1, [1115].log_data[3].valid := 1, [1115].log_data[4].valid := 1, [1115].time.Year := 2022, [1115].time.Month := 4, [1115].time.Day := 27, [1115].time.Hour := 18, [1115].time.Minute := 29, [1115].time.Second := 59, [1115].time.DST_ON := 1, [1116].log_data[0].min := 1.0,
        [1116].log_data[0].max := 1.0, [1116].log_data[0].total := 300.0, [1116].log_data[0].time := 300.0, [1116].log_data[0].minminute := 30, [1116].log_data[0].maxminute := 30, [1116].log_data[0].valid := 1, [1116].log_data[1].valid := 1, [1116].log_data[2].valid := 1, [1116].log_data[3].valid := 1, [1116].log_data[4].valid := 1, [1116].time.Year := 2022, [1116].time.Month := 4, [1116].time.Day := 27, [1116].time.Hour := 18, [1116].time.Minute := 34, [1116].time.Second := 59, [1116].time.DST_ON := 1, [1117].log_data[0].min := 1.0, [1117].log_data[0].max := 1.0, [1117].log_data[0].total := 300.0, [1117].log_data[0].time := 300.0, [1117].log_data[0].minminute := 35, [1117].log_data[0].maxminute := 35, [1117].log_data[0].valid := 1, [1117].log_data[1].valid := 1, [1117].log_data[2].valid := 1, [1117].log_data[3].valid := 1, [1117].log_data[4].valid := 1, [1117].time.Year := 2022, [1117].time.Month := 4, [1117].time.Day := 27, [1117].time.Hour := 18, [1117].time.Minute := 39, [1117].time.Second := 59, [1117].time.DST_ON := 1, [1118].log_data[0].min := 1.0, [1118].log_data[0].max := 1.0, [1118].log_data[0].total := 300.0, [1118].log_data[0].time := 300.0, [1118].log_data[0].minminute := 40, [1118].log_data[0].maxminute := 40, [1118].log_data[0].valid := 1, [1118].log_data[1].valid := 1, [1118].log_data[2].valid := 1, [1118].log_data[3].valid := 1, [1118].log_data[4].valid := 1, [1118].time.Year := 2022, [1118].time.Month := 4, [1118].time.Day := 27, [1118].time.Hour := 18, [1118].time.Minute := 44, [1118].time.Second := 59, [1118].time.DST_ON := 1, [1119].log_data[0].min := 1.0, [1119].log_data[0].max := 1.0, [1119].log_data[0].total := 300.0, [1119].log_data[0].time := 300.0, [1119].log_data[0].minminute := 45, [1119].log_data[0].maxminute := 45, [1119].log_data[0].valid := 1,
        [1119].log_data[1].valid := 1, [1119].log_data[2].valid := 1, [1119].log_data[3].valid := 1, [1119].log_data[4].valid := 1, [1119].time.Year := 2022, [1119].time.Month := 4, [1119].time.Day := 27, [1119].time.Hour := 18, [1119].time.Minute := 49, [1119].time.Second := 59, [1119].time.DST_ON := 1, [1120].log_data[0].min := 1.0, [1120].log_data[0].max := 1.0, [1120].log_data[0].total := 300.0, [1120].log_data[0].time := 300.0, [1120].log_data[0].minminute := 50, [1120].log_data[0].maxminute := 50, [1120].log_data[0].valid := 1, [1120].log_data[1].valid := 1, [1120].log_data[2].valid := 1, [1120].log_data[3].valid := 1, [1120].log_data[4].valid := 1, [1120].time.Year := 2022, [1120].time.Month := 4, [1120].time.Day := 27, [1120].time.Hour := 18, [1120].time.Minute := 54, [1120].time.Second := 59, [1120].time.DST_ON := 1, [1121].log_data[0].min := 1.0, [1121].log_data[0].max := 1.0, [1121].log_data[0].total := 300.0, [1121].log_data[0].time := 300.0, [1121].log_data[0].minminute := 55, [1121].log_data[0].maxminute := 55, [1121].log_data[0].valid := 1, [1121].log_data[1].valid := 1, [1121].log_data[2].valid := 1, [1121].log_data[3].valid := 1, [1121].log_data[4].valid := 1, [1121].time.Year := 2022, [1121].time.Month := 4, [1121].time.Day := 27, [1121].time.Hour := 18, [1121].time.Minute := 59, [1121].time.Second := 59, [1121].time.DST_ON := 1, [1122].log_data[0].min := 1.0, [1122].log_data[0].max := 1.0, [1122].log_data[0].total := 300.0, [1122].log_data[0].time := 300.0, [1122].log_data[0].valid := 1, [1122].log_data[1].valid := 1, [1122].log_data[2].valid := 1, [1122].log_data[3].valid := 1, [1122].log_data[4].valid := 1, [1122].time.Year := 2022, [1122].time.Month := 4, [1122].time.Day := 27, [1122].time.Hour := 19,
        [1122].time.Minute := 4, [1122].time.Second := 59, [1122].time.DST_ON := 1, [1123].log_data[0].min := 1.0, [1123].log_data[0].max := 1.0, [1123].log_data[0].total := 300.0, [1123].log_data[0].time := 300.0, [1123].log_data[0].minminute := 5, [1123].log_data[0].maxminute := 5, [1123].log_data[0].valid := 1, [1123].log_data[1].valid := 1, [1123].log_data[2].valid := 1, [1123].log_data[3].valid := 1, [1123].log_data[4].valid := 1, [1123].time.Year := 2022, [1123].time.Month := 4, [1123].time.Day := 27, [1123].time.Hour := 19, [1123].time.Minute := 9, [1123].time.Second := 59, [1123].time.DST_ON := 1, [1124].log_data[0].min := 1.0, [1124].log_data[0].max := 1.0, [1124].log_data[0].total := 299.999, [1124].log_data[0].time := 299.999, [1124].log_data[0].minminute := 10, [1124].log_data[0].maxminute := 10, [1124].log_data[0].valid := 1, [1124].log_data[1].valid := 1, [1124].log_data[2].valid := 1, [1124].log_data[3].valid := 1, [1124].log_data[4].valid := 1, [1124].time.Year := 2022, [1124].time.Month := 4, [1124].time.Day := 27, [1124].time.Hour := 19, [1124].time.Minute := 14, [1124].time.Second := 59, [1124].time.DST_ON := 1, [1125].log_data[0].min := 1.0, [1125].log_data[0].max := 1.0, [1125].log_data[0].total := 300.0, [1125].log_data[0].time := 300.0, [1125].log_data[0].minminute := 15, [1125].log_data[0].maxminute := 15, [1125].log_data[0].valid := 1, [1125].log_data[1].valid := 1, [1125].log_data[2].valid := 1, [1125].log_data[3].valid := 1, [1125].log_data[4].valid := 1, [1125].time.Year := 2022, [1125].time.Month := 4, [1125].time.Day := 27, [1125].time.Hour := 19, [1125].time.Minute := 19, [1125].time.Second := 59, [1125].time.DST_ON := 1, [1126].log_data[0].min := 1.0, [1126].log_data[0].max := 1.0, [1126].log_data[0].total := 300.0,
        [1126].log_data[0].time := 300.0, [1126].log_data[0].minminute := 20, [1126].log_data[0].maxminute := 20, [1126].log_data[0].valid := 1, [1126].log_data[1].valid := 1, [1126].log_data[2].valid := 1, [1126].log_data[3].valid := 1, [1126].log_data[4].valid := 1, [1126].time.Year := 2022, [1126].time.Month := 4, [1126].time.Day := 27, [1126].time.Hour := 19, [1126].time.Minute := 24, [1126].time.Second := 59, [1126].time.DST_ON := 1, [1127].log_data[0].min := 1.0, [1127].log_data[0].max := 1.0, [1127].log_data[0].total := 300.0, [1127].log_data[0].time := 300.0, [1127].log_data[0].minminute := 25, [1127].log_data[0].maxminute := 25, [1127].log_data[0].valid := 1, [1127].log_data[1].valid := 1, [1127].log_data[2].valid := 1, [1127].log_data[3].valid := 1, [1127].log_data[4].valid := 1, [1127].time.Year := 2022, [1127].time.Month := 4, [1127].time.Day := 27, [1127].time.Hour := 19, [1127].time.Minute := 29, [1127].time.Second := 59, [1127].time.DST_ON := 1, [1128].log_data[0].min := 1.0, [1128].log_data[0].max := 1.0, [1128].log_data[0].total := 300.0, [1128].log_data[0].time := 300.0, [1128].log_data[0].minminute := 30, [1128].log_data[0].maxminute := 30, [1128].log_data[0].valid := 1, [1128].log_data[1].valid := 1, [1128].log_data[2].valid := 1, [1128].log_data[3].valid := 1, [1128].log_data[4].valid := 1, [1128].time.Year := 2022, [1128].time.Month := 4, [1128].time.Day := 27, [1128].time.Hour := 19, [1128].time.Minute := 34, [1128].time.Second := 59, [1128].time.DST_ON := 1, [1129].log_data[0].min := 1.0, [1129].log_data[0].max := 1.0, [1129].log_data[0].total := 300.0, [1129].log_data[0].time := 300.0, [1129].log_data[0].minminute := 35, [1129].log_data[0].maxminute := 35, [1129].log_data[0].valid := 1, [1129].log_data[1].valid := 1, [1129].log_data[2].valid := 1,
        [1129].log_data[3].valid := 1, [1129].log_data[4].valid := 1, [1129].time.Year := 2022, [1129].time.Month := 4, [1129].time.Day := 27, [1129].time.Hour := 19, [1129].time.Minute := 39, [1129].time.Second := 59, [1129].time.DST_ON := 1, [1130].log_data[0].min := 1.0, [1130].log_data[0].max := 1.0, [1130].log_data[0].total := 300.0, [1130].log_data[0].time := 300.0, [1130].log_data[0].minminute := 40, [1130].log_data[0].maxminute := 40, [1130].log_data[0].valid := 1, [1130].log_data[1].valid := 1, [1130].log_data[2].valid := 1, [1130].log_data[3].valid := 1, [1130].log_data[4].valid := 1, [1130].time.Year := 2022, [1130].time.Month := 4, [1130].time.Day := 27, [1130].time.Hour := 19, [1130].time.Minute := 44, [1130].time.Second := 59, [1130].time.DST_ON := 1, [1131].log_data[0].min := 1.0, [1131].log_data[0].max := 1.0, [1131].log_data[0].total := 300.0, [1131].log_data[0].time := 300.0, [1131].log_data[0].minminute := 45, [1131].log_data[0].maxminute := 45, [1131].log_data[0].valid := 1, [1131].log_data[1].valid := 1, [1131].log_data[2].valid := 1, [1131].log_data[3].valid := 1, [1131].log_data[4].valid := 1, [1131].time.Year := 2022, [1131].time.Month := 4, [1131].time.Day := 27, [1131].time.Hour := 19, [1131].time.Minute := 49, [1131].time.Second := 59, [1131].time.DST_ON := 1, [1132].log_data[0].min := 1.0, [1132].log_data[0].max := 1.0, [1132].log_data[0].total := 300.0, [1132].log_data[0].time := 300.0, [1132].log_data[0].minminute := 50, [1132].log_data[0].maxminute := 50, [1132].log_data[0].valid := 1, [1132].log_data[1].valid := 1, [1132].log_data[2].valid := 1, [1132].log_data[3].valid := 1, [1132].log_data[4].valid := 1, [1132].time.Year := 2022, [1132].time.Month := 4, [1132].time.Day := 27, [1132].time.Hour := 19,
        [1132].time.Minute := 54, [1132].time.Second := 59, [1132].time.DST_ON := 1, [1133].log_data[0].min := 1.0, [1133].log_data[0].max := 1.0, [1133].log_data[0].total := 300.0, [1133].log_data[0].time := 300.0, [1133].log_data[0].minminute := 55, [1133].log_data[0].maxminute := 55, [1133].log_data[0].valid := 1, [1133].log_data[1].valid := 1, [1133].log_data[2].valid := 1, [1133].log_data[3].valid := 1, [1133].log_data[4].valid := 1, [1133].time.Year := 2022, [1133].time.Month := 4, [1133].time.Day := 27, [1133].time.Hour := 19, [1133].time.Minute := 59, [1133].time.Second := 59, [1133].time.DST_ON := 1, [1134].log_data[0].min := 1.0, [1134].log_data[0].max := 1.0, [1134].log_data[0].total := 300.0, [1134].log_data[0].time := 300.0, [1134].log_data[0].valid := 1, [1134].log_data[1].valid := 1, [1134].log_data[2].valid := 1, [1134].log_data[3].valid := 1, [1134].log_data[4].valid := 1, [1134].time.Year := 2022, [1134].time.Month := 4, [1134].time.Day := 27, [1134].time.Hour := 20, [1134].time.Minute := 4, [1134].time.Second := 59, [1134].time.DST_ON := 1, [1135].log_data[0].min := 1.0, [1135].log_data[0].max := 1.0, [1135].log_data[0].total := 300.0, [1135].log_data[0].time := 300.0, [1135].log_data[0].minminute := 5, [1135].log_data[0].maxminute := 5, [1135].log_data[0].valid := 1, [1135].log_data[1].valid := 1, [1135].log_data[2].valid := 1, [1135].log_data[3].valid := 1, [1135].log_data[4].valid := 1, [1135].time.Year := 2022, [1135].time.Month := 4, [1135].time.Day := 27, [1135].time.Hour := 20, [1135].time.Minute := 9, [1135].time.Second := 59, [1135].time.DST_ON := 1, [1136].log_data[0].min := 1.0, [1136].log_data[0].max := 1.0, [1136].log_data[0].total := 299.999, [1136].log_data[0].time := 299.999, [1136].log_data[0].minminute := 10,
        [1136].log_data[0].maxminute := 10, [1136].log_data[0].valid := 1, [1136].log_data[1].valid := 1, [1136].log_data[2].valid := 1, [1136].log_data[3].valid := 1, [1136].log_data[4].valid := 1, [1136].time.Year := 2022, [1136].time.Month := 4, [1136].time.Day := 27, [1136].time.Hour := 20, [1136].time.Minute := 14, [1136].time.Second := 59, [1136].time.DST_ON := 1, [1137].log_data[0].min := 1.0, [1137].log_data[0].max := 1.0, [1137].log_data[0].total := 300.0, [1137].log_data[0].time := 300.0, [1137].log_data[0].minminute := 15, [1137].log_data[0].maxminute := 15, [1137].log_data[0].valid := 1, [1137].log_data[1].valid := 1, [1137].log_data[2].valid := 1, [1137].log_data[3].valid := 1, [1137].log_data[4].valid := 1, [1137].time.Year := 2022, [1137].time.Month := 4, [1137].time.Day := 27, [1137].time.Hour := 20, [1137].time.Minute := 19, [1137].time.Second := 59, [1137].time.DST_ON := 1, [1138].log_data[0].min := 1.0, [1138].log_data[0].max := 1.0, [1138].log_data[0].total := 300.0, [1138].log_data[0].time := 300.0, [1138].log_data[0].minminute := 20, [1138].log_data[0].maxminute := 20, [1138].log_data[0].valid := 1, [1138].log_data[1].valid := 1, [1138].log_data[2].valid := 1, [1138].log_data[3].valid := 1, [1138].log_data[4].valid := 1, [1138].time.Year := 2022, [1138].time.Month := 4, [1138].time.Day := 27, [1138].time.Hour := 20, [1138].time.Minute := 24, [1138].time.Second := 59, [1138].time.DST_ON := 1, [1139].log_data[0].min := 1.0, [1139].log_data[0].max := 1.0, [1139].log_data[0].total := 300.0, [1139].log_data[0].time := 300.0, [1139].log_data[0].minminute := 25, [1139].log_data[0].maxminute := 25, [1139].log_data[0].valid := 1, [1139].log_data[1].valid := 1, [1139].log_data[2].valid := 1, [1139].log_data[3].valid := 1, [1139].log_data[4].valid := 1,
        [1139].time.Year := 2022, [1139].time.Month := 4, [1139].time.Day := 27, [1139].time.Hour := 20, [1139].time.Minute := 29, [1139].time.Second := 59, [1139].time.DST_ON := 1, [1140].log_data[0].min := 1.0, [1140].log_data[0].max := 1.0, [1140].log_data[0].total := 300.0, [1140].log_data[0].time := 300.0, [1140].log_data[0].minminute := 30, [1140].log_data[0].maxminute := 30, [1140].log_data[0].valid := 1, [1140].log_data[1].valid := 1, [1140].log_data[2].valid := 1, [1140].log_data[3].valid := 1, [1140].log_data[4].valid := 1, [1140].time.Year := 2022, [1140].time.Month := 4, [1140].time.Day := 27, [1140].time.Hour := 20, [1140].time.Minute := 34, [1140].time.Second := 59, [1140].time.DST_ON := 1, [1141].log_data[0].min := 1.0, [1141].log_data[0].max := 1.0, [1141].log_data[0].total := 300.0, [1141].log_data[0].time := 300.0, [1141].log_data[0].minminute := 35, [1141].log_data[0].maxminute := 35, [1141].log_data[0].valid := 1, [1141].log_data[1].valid := 1, [1141].log_data[2].valid := 1, [1141].log_data[3].valid := 1, [1141].log_data[4].valid := 1, [1141].time.Year := 2022, [1141].time.Month := 4, [1141].time.Day := 27, [1141].time.Hour := 20, [1141].time.Minute := 39, [1141].time.Second := 59, [1141].time.DST_ON := 1, [1142].log_data[0].min := 1.0, [1142].log_data[0].max := 1.0, [1142].log_data[0].total := 300.0, [1142].log_data[0].time := 300.0, [1142].log_data[0].minminute := 40, [1142].log_data[0].maxminute := 40, [1142].log_data[0].valid := 1, [1142].log_data[1].valid := 1, [1142].log_data[2].valid := 1, [1142].log_data[3].valid := 1, [1142].log_data[4].valid := 1, [1142].time.Year := 2022, [1142].time.Month := 4, [1142].time.Day := 27, [1142].time.Hour := 20, [1142].time.Minute := 44, [1142].time.Second := 59,
        [1142].time.DST_ON := 1, [1143].log_data[0].min := 1.0, [1143].log_data[0].max := 1.0, [1143].log_data[0].total := 300.0, [1143].log_data[0].time := 300.0, [1143].log_data[0].minminute := 45, [1143].log_data[0].maxminute := 45, [1143].log_data[0].valid := 1, [1143].log_data[1].valid := 1, [1143].log_data[2].valid := 1, [1143].log_data[3].valid := 1, [1143].log_data[4].valid := 1, [1143].time.Year := 2022, [1143].time.Month := 4, [1143].time.Day := 27, [1143].time.Hour := 20, [1143].time.Minute := 49, [1143].time.Second := 59, [1143].time.DST_ON := 1, [1144].log_data[0].min := 1.0, [1144].log_data[0].max := 1.0, [1144].log_data[0].total := 300.0, [1144].log_data[0].time := 300.0, [1144].log_data[0].minminute := 50, [1144].log_data[0].maxminute := 50, [1144].log_data[0].valid := 1, [1144].log_data[1].valid := 1, [1144].log_data[2].valid := 1, [1144].log_data[3].valid := 1, [1144].log_data[4].valid := 1, [1144].time.Year := 2022, [1144].time.Month := 4, [1144].time.Day := 27, [1144].time.Hour := 20, [1144].time.Minute := 54, [1144].time.Second := 59, [1144].time.DST_ON := 1, [1145].log_data[0].min := 1.0, [1145].log_data[0].max := 1.0, [1145].log_data[0].total := 300.0, [1145].log_data[0].time := 300.0, [1145].log_data[0].minminute := 55, [1145].log_data[0].maxminute := 55, [1145].log_data[0].valid := 1, [1145].log_data[1].valid := 1, [1145].log_data[2].valid := 1, [1145].log_data[3].valid := 1, [1145].log_data[4].valid := 1, [1145].time.Year := 2022, [1145].time.Month := 4, [1145].time.Day := 27, [1145].time.Hour := 20, [1145].time.Minute := 59, [1145].time.Second := 59, [1145].time.DST_ON := 1, [1146].log_data[0].min := 1.0, [1146].log_data[0].max := 1.0, [1146].log_data[0].total := 300.0, [1146].log_data[0].time := 300.0, [1146].log_data[0].valid := 1,
        [1146].log_data[1].valid := 1, [1146].log_data[2].valid := 1, [1146].log_data[3].valid := 1, [1146].log_data[4].valid := 1, [1146].time.Year := 2022, [1146].time.Month := 4, [1146].time.Day := 27, [1146].time.Hour := 21, [1146].time.Minute := 4, [1146].time.Second := 59, [1146].time.DST_ON := 1, [1147].log_data[0].min := 1.0, [1147].log_data[0].max := 1.0, [1147].log_data[0].total := 300.0, [1147].log_data[0].time := 300.0, [1147].log_data[0].minminute := 5, [1147].log_data[0].maxminute := 5, [1147].log_data[0].valid := 1, [1147].log_data[1].valid := 1, [1147].log_data[2].valid := 1, [1147].log_data[3].valid := 1, [1147].log_data[4].valid := 1, [1147].time.Year := 2022, [1147].time.Month := 4, [1147].time.Day := 27, [1147].time.Hour := 21, [1147].time.Minute := 9, [1147].time.Second := 59, [1147].time.DST_ON := 1, [1148].log_data[0].min := 1.0, [1148].log_data[0].max := 1.0, [1148].log_data[0].total := 300.0, [1148].log_data[0].time := 300.0, [1148].log_data[0].minminute := 10, [1148].log_data[0].maxminute := 10, [1148].log_data[0].valid := 1, [1148].log_data[1].valid := 1, [1148].log_data[2].valid := 1, [1148].log_data[3].valid := 1, [1148].log_data[4].valid := 1, [1148].time.Year := 2022, [1148].time.Month := 4, [1148].time.Day := 27, [1148].time.Hour := 21, [1148].time.Minute := 14, [1148].time.Second := 59, [1148].time.DST_ON := 1, [1149].log_data[0].min := 1.0, [1149].log_data[0].max := 1.0, [1149].log_data[0].total := 300.0, [1149].log_data[0].time := 300.0, [1149].log_data[0].minminute := 15, [1149].log_data[0].maxminute := 15, [1149].log_data[0].valid := 1, [1149].log_data[1].valid := 1, [1149].log_data[2].valid := 1, [1149].log_data[3].valid := 1, [1149].log_data[4].valid := 1, [1149].time.Year := 2022, [1149].time.Month := 4,
        [1149].time.Day := 27, [1149].time.Hour := 21, [1149].time.Minute := 19, [1149].time.Second := 59, [1149].time.DST_ON := 1, [1150].log_data[0].min := 1.0, [1150].log_data[0].max := 1.0, [1150].log_data[0].total := 300.0, [1150].log_data[0].time := 300.0, [1150].log_data[0].minminute := 20, [1150].log_data[0].maxminute := 20, [1150].log_data[0].valid := 1, [1150].log_data[1].valid := 1, [1150].log_data[2].valid := 1, [1150].log_data[3].valid := 1, [1150].log_data[4].valid := 1, [1150].time.Year := 2022, [1150].time.Month := 4, [1150].time.Day := 27, [1150].time.Hour := 21, [1150].time.Minute := 24, [1150].time.Second := 59, [1150].time.DST_ON := 1, [1151].log_data[0].min := 1.0, [1151].log_data[0].max := 1.0, [1151].log_data[0].total := 300.0, [1151].log_data[0].time := 300.0, [1151].log_data[0].minminute := 25, [1151].log_data[0].maxminute := 25, [1151].log_data[0].valid := 1, [1151].log_data[1].valid := 1, [1151].log_data[2].valid := 1, [1151].log_data[3].valid := 1, [1151].log_data[4].valid := 1, [1151].time.Year := 2022, [1151].time.Month := 4, [1151].time.Day := 27, [1151].time.Hour := 21, [1151].time.Minute := 29, [1151].time.Second := 59, [1151].time.DST_ON := 1, [1152].log_data[0].min := 1.0, [1152].log_data[0].max := 1.0, [1152].log_data[0].total := 300.0, [1152].log_data[0].time := 300.0, [1152].log_data[0].minminute := 30, [1152].log_data[0].maxminute := 30, [1152].log_data[0].valid := 1, [1152].log_data[1].valid := 1, [1152].log_data[2].valid := 1, [1152].log_data[3].valid := 1, [1152].log_data[4].valid := 1, [1152].time.Year := 2022, [1152].time.Month := 4, [1152].time.Day := 27, [1152].time.Hour := 21, [1152].time.Minute := 34, [1152].time.Second := 59, [1152].time.DST_ON := 1, [1153].log_data[0].min := 1.0,
        [1153].log_data[0].max := 1.0, [1153].log_data[0].total := 300.0, [1153].log_data[0].time := 300.0, [1153].log_data[0].minminute := 35, [1153].log_data[0].maxminute := 35, [1153].log_data[0].valid := 1, [1153].log_data[1].valid := 1, [1153].log_data[2].valid := 1, [1153].log_data[3].valid := 1, [1153].log_data[4].valid := 1, [1153].time.Year := 2022, [1153].time.Month := 4, [1153].time.Day := 27, [1153].time.Hour := 21, [1153].time.Minute := 39, [1153].time.Second := 59, [1153].time.DST_ON := 1, [1154].log_data[0].min := 1.0, [1154].log_data[0].max := 1.0, [1154].log_data[0].total := 300.0, [1154].log_data[0].time := 300.0, [1154].log_data[0].minminute := 40, [1154].log_data[0].maxminute := 40, [1154].log_data[0].valid := 1, [1154].log_data[1].valid := 1, [1154].log_data[2].valid := 1, [1154].log_data[3].valid := 1, [1154].log_data[4].valid := 1, [1154].time.Year := 2022, [1154].time.Month := 4, [1154].time.Day := 27, [1154].time.Hour := 21, [1154].time.Minute := 44, [1154].time.Second := 59, [1154].time.DST_ON := 1, [1155].log_data[0].min := 1.0, [1155].log_data[0].max := 1.0, [1155].log_data[0].total := 300.0, [1155].log_data[0].time := 300.0, [1155].log_data[0].minminute := 45, [1155].log_data[0].maxminute := 45, [1155].log_data[0].valid := 1, [1155].log_data[1].valid := 1, [1155].log_data[2].valid := 1, [1155].log_data[3].valid := 1, [1155].log_data[4].valid := 1, [1155].time.Year := 2022, [1155].time.Month := 4, [1155].time.Day := 27, [1155].time.Hour := 21, [1155].time.Minute := 49, [1155].time.Second := 59, [1155].time.DST_ON := 1, [1156].log_data[0].min := 1.0, [1156].log_data[0].max := 1.0, [1156].log_data[0].total := 300.0, [1156].log_data[0].time := 300.0, [1156].log_data[0].minminute := 50, [1156].log_data[0].maxminute := 50, [1156].log_data[0].valid := 1,
        [1156].log_data[1].valid := 1, [1156].log_data[2].valid := 1, [1156].log_data[3].valid := 1, [1156].log_data[4].valid := 1, [1156].time.Year := 2022, [1156].time.Month := 4, [1156].time.Day := 27, [1156].time.Hour := 21, [1156].time.Minute := 54, [1156].time.Second := 59, [1156].time.DST_ON := 1, [1157].log_data[0].min := 1.0, [1157].log_data[0].max := 1.0, [1157].log_data[0].total := 300.0, [1157].log_data[0].time := 300.0, [1157].log_data[0].minminute := 55, [1157].log_data[0].maxminute := 55, [1157].log_data[0].valid := 1, [1157].log_data[1].valid := 1, [1157].log_data[2].valid := 1, [1157].log_data[3].valid := 1, [1157].log_data[4].valid := 1, [1157].time.Year := 2022, [1157].time.Month := 4, [1157].time.Day := 27, [1157].time.Hour := 21, [1157].time.Minute := 59, [1157].time.Second := 59, [1157].time.DST_ON := 1, [1158].log_data[0].min := 1.0, [1158].log_data[0].max := 1.0, [1158].log_data[0].total := 300.0, [1158].log_data[0].time := 300.0, [1158].log_data[0].valid := 1, [1158].log_data[1].valid := 1, [1158].log_data[2].valid := 1, [1158].log_data[3].valid := 1, [1158].log_data[4].valid := 1, [1158].time.Year := 2022, [1158].time.Month := 4, [1158].time.Day := 27, [1158].time.Hour := 22, [1158].time.Minute := 4, [1158].time.Second := 59, [1158].time.DST_ON := 1, [1159].log_data[0].min := 1.0, [1159].log_data[0].max := 1.0, [1159].log_data[0].total := 300.0, [1159].log_data[0].time := 300.0, [1159].log_data[0].minminute := 5, [1159].log_data[0].maxminute := 5, [1159].log_data[0].valid := 1, [1159].log_data[1].valid := 1, [1159].log_data[2].valid := 1, [1159].log_data[3].valid := 1, [1159].log_data[4].valid := 1, [1159].time.Year := 2022, [1159].time.Month := 4, [1159].time.Day := 27, [1159].time.Hour := 22,
        [1159].time.Minute := 9, [1159].time.Second := 59, [1159].time.DST_ON := 1, [1160].log_data[0].min := 1.0, [1160].log_data[0].max := 1.0, [1160].log_data[0].total := 300.0, [1160].log_data[0].time := 300.0, [1160].log_data[0].minminute := 10, [1160].log_data[0].maxminute := 10, [1160].log_data[0].valid := 1, [1160].log_data[1].valid := 1, [1160].log_data[2].valid := 1, [1160].log_data[3].valid := 1, [1160].log_data[4].valid := 1, [1160].time.Year := 2022, [1160].time.Month := 4, [1160].time.Day := 27, [1160].time.Hour := 22, [1160].time.Minute := 14, [1160].time.Second := 59, [1160].time.DST_ON := 1, [1161].log_data[0].min := 1.0, [1161].log_data[0].max := 1.0, [1161].log_data[0].total := 300.0, [1161].log_data[0].time := 300.0, [1161].log_data[0].minminute := 15, [1161].log_data[0].maxminute := 15, [1161].log_data[0].valid := 1, [1161].log_data[1].valid := 1, [1161].log_data[2].valid := 1, [1161].log_data[3].valid := 1, [1161].log_data[4].valid := 1, [1161].time.Year := 2022, [1161].time.Month := 4, [1161].time.Day := 27, [1161].time.Hour := 22, [1161].time.Minute := 19, [1161].time.Second := 59, [1161].time.DST_ON := 1, [1162].log_data[0].min := 1.0, [1162].log_data[0].max := 1.0, [1162].log_data[0].total := 300.0, [1162].log_data[0].time := 300.0, [1162].log_data[0].minminute := 20, [1162].log_data[0].maxminute := 20, [1162].log_data[0].valid := 1, [1162].log_data[1].valid := 1, [1162].log_data[2].valid := 1, [1162].log_data[3].valid := 1, [1162].log_data[4].valid := 1, [1162].time.Year := 2022, [1162].time.Month := 4, [1162].time.Day := 27, [1162].time.Hour := 22, [1162].time.Minute := 24, [1162].time.Second := 59, [1162].time.DST_ON := 1, [1163].log_data[0].min := 1.0, [1163].log_data[0].max := 1.0, [1163].log_data[0].total := 300.0,
        [1163].log_data[0].time := 300.0, [1163].log_data[0].minminute := 25, [1163].log_data[0].maxminute := 25, [1163].log_data[0].valid := 1, [1163].log_data[1].valid := 1, [1163].log_data[2].valid := 1, [1163].log_data[3].valid := 1, [1163].log_data[4].valid := 1, [1163].time.Year := 2022, [1163].time.Month := 4, [1163].time.Day := 27, [1163].time.Hour := 22, [1163].time.Minute := 29, [1163].time.Second := 59, [1163].time.DST_ON := 1, [1164].log_data[0].min := 1.0, [1164].log_data[0].max := 1.0, [1164].log_data[0].total := 300.0, [1164].log_data[0].time := 300.0, [1164].log_data[0].minminute := 30, [1164].log_data[0].maxminute := 30, [1164].log_data[0].valid := 1, [1164].log_data[1].valid := 1, [1164].log_data[2].valid := 1, [1164].log_data[3].valid := 1, [1164].log_data[4].valid := 1, [1164].time.Year := 2022, [1164].time.Month := 4, [1164].time.Day := 27, [1164].time.Hour := 22, [1164].time.Minute := 34, [1164].time.Second := 59, [1164].time.DST_ON := 1, [1165].log_data[0].min := 1.0, [1165].log_data[0].max := 1.0, [1165].log_data[0].total := 300.0, [1165].log_data[0].time := 300.0, [1165].log_data[0].minminute := 35, [1165].log_data[0].maxminute := 35, [1165].log_data[0].valid := 1, [1165].log_data[1].valid := 1, [1165].log_data[2].valid := 1, [1165].log_data[3].valid := 1, [1165].log_data[4].valid := 1, [1165].time.Year := 2022, [1165].time.Month := 4, [1165].time.Day := 27, [1165].time.Hour := 22, [1165].time.Minute := 39, [1165].time.Second := 59, [1165].time.DST_ON := 1, [1166].log_data[0].min := 1.0, [1166].log_data[0].max := 1.0, [1166].log_data[0].total := 300.0, [1166].log_data[0].time := 300.0, [1166].log_data[0].minminute := 40, [1166].log_data[0].maxminute := 40, [1166].log_data[0].valid := 1, [1166].log_data[1].valid := 1, [1166].log_data[2].valid := 1,
        [1166].log_data[3].valid := 1, [1166].log_data[4].valid := 1, [1166].time.Year := 2022, [1166].time.Month := 4, [1166].time.Day := 27, [1166].time.Hour := 22, [1166].time.Minute := 44, [1166].time.Second := 59, [1166].time.DST_ON := 1, [1167].log_data[0].min := 1.0, [1167].log_data[0].max := 1.0, [1167].log_data[0].total := 300.0, [1167].log_data[0].time := 300.0, [1167].log_data[0].minminute := 45, [1167].log_data[0].maxminute := 45, [1167].log_data[0].valid := 1, [1167].log_data[1].valid := 1, [1167].log_data[2].valid := 1, [1167].log_data[3].valid := 1, [1167].log_data[4].valid := 1, [1167].time.Year := 2022, [1167].time.Month := 4, [1167].time.Day := 27, [1167].time.Hour := 22, [1167].time.Minute := 49, [1167].time.Second := 59, [1167].time.DST_ON := 1, [1168].log_data[0].min := 1.0, [1168].log_data[0].max := 1.0, [1168].log_data[0].total := 300.0, [1168].log_data[0].time := 300.0, [1168].log_data[0].minminute := 50, [1168].log_data[0].maxminute := 50, [1168].log_data[0].valid := 1, [1168].log_data[1].valid := 1, [1168].log_data[2].valid := 1, [1168].log_data[3].valid := 1, [1168].log_data[4].valid := 1, [1168].time.Year := 2022, [1168].time.Month := 4, [1168].time.Day := 27, [1168].time.Hour := 22, [1168].time.Minute := 54, [1168].time.Second := 59, [1168].time.DST_ON := 1, [1169].log_data[0].min := 1.0, [1169].log_data[0].max := 1.0, [1169].log_data[0].total := 300.0, [1169].log_data[0].time := 300.0, [1169].log_data[0].minminute := 55, [1169].log_data[0].maxminute := 55, [1169].log_data[0].valid := 1, [1169].log_data[1].valid := 1, [1169].log_data[2].valid := 1, [1169].log_data[3].valid := 1, [1169].log_data[4].valid := 1, [1169].time.Year := 2022, [1169].time.Month := 4, [1169].time.Day := 27, [1169].time.Hour := 22,
        [1169].time.Minute := 59, [1169].time.Second := 59, [1169].time.DST_ON := 1, [1170].log_data[0].min := 1.0, [1170].log_data[0].max := 1.0, [1170].log_data[0].total := 300.0, [1170].log_data[0].time := 300.0, [1170].log_data[0].valid := 1, [1170].log_data[1].valid := 1, [1170].log_data[2].valid := 1, [1170].log_data[3].valid := 1, [1170].log_data[4].valid := 1, [1170].time.Year := 2022, [1170].time.Month := 4, [1170].time.Day := 27, [1170].time.Hour := 23, [1170].time.Minute := 4, [1170].time.Second := 59, [1170].time.DST_ON := 1, [1171].log_data[0].min := 1.0, [1171].log_data[0].max := 1.0, [1171].log_data[0].total := 300.0, [1171].log_data[0].time := 300.0, [1171].log_data[0].minminute := 5, [1171].log_data[0].maxminute := 5, [1171].log_data[0].valid := 1, [1171].log_data[1].valid := 1, [1171].log_data[2].valid := 1, [1171].log_data[3].valid := 1, [1171].log_data[4].valid := 1, [1171].time.Year := 2022, [1171].time.Month := 4, [1171].time.Day := 27, [1171].time.Hour := 23, [1171].time.Minute := 9, [1171].time.Second := 59, [1171].time.DST_ON := 1, [1172].log_data[0].min := 1.0, [1172].log_data[0].max := 1.0, [1172].log_data[0].total := 300.0, [1172].log_data[0].time := 300.0, [1172].log_data[0].minminute := 10, [1172].log_data[0].maxminute := 10, [1172].log_data[0].valid := 1, [1172].log_data[1].valid := 1, [1172].log_data[2].valid := 1, [1172].log_data[3].valid := 1, [1172].log_data[4].valid := 1, [1172].time.Year := 2022, [1172].time.Month := 4, [1172].time.Day := 27, [1172].time.Hour := 23, [1172].time.Minute := 14, [1172].time.Second := 59, [1172].time.DST_ON := 1, [1173].log_data[0].min := 1.0, [1173].log_data[0].max := 1.0, [1173].log_data[0].total := 300.0, [1173].log_data[0].time := 300.0, [1173].log_data[0].minminute := 15,
        [1173].log_data[0].maxminute := 15, [1173].log_data[0].valid := 1, [1173].log_data[1].valid := 1, [1173].log_data[2].valid := 1, [1173].log_data[3].valid := 1, [1173].log_data[4].valid := 1, [1173].time.Year := 2022, [1173].time.Month := 4, [1173].time.Day := 27, [1173].time.Hour := 23, [1173].time.Minute := 19, [1173].time.Second := 59, [1173].time.DST_ON := 1, [1174].log_data[0].min := 1.0, [1174].log_data[0].max := 1.0, [1174].log_data[0].total := 299.999, [1174].log_data[0].time := 299.999, [1174].log_data[0].minminute := 20, [1174].log_data[0].maxminute := 20, [1174].log_data[0].valid := 1, [1174].log_data[1].valid := 1, [1174].log_data[2].valid := 1, [1174].log_data[3].valid := 1, [1174].log_data[4].valid := 1, [1174].time.Year := 2022, [1174].time.Month := 4, [1174].time.Day := 27, [1174].time.Hour := 23, [1174].time.Minute := 24, [1174].time.Second := 59, [1174].time.DST_ON := 1, [1175].log_data[0].min := 1.0, [1175].log_data[0].max := 1.0, [1175].log_data[0].total := 300.0, [1175].log_data[0].time := 300.0, [1175].log_data[0].minminute := 25, [1175].log_data[0].maxminute := 25, [1175].log_data[0].valid := 1, [1175].log_data[1].valid := 1, [1175].log_data[2].valid := 1, [1175].log_data[3].valid := 1, [1175].log_data[4].valid := 1, [1175].time.Year := 2022, [1175].time.Month := 4, [1175].time.Day := 27, [1175].time.Hour := 23, [1175].time.Minute := 29, [1175].time.Second := 59, [1175].time.DST_ON := 1, [1176].log_data[0].min := 1.0, [1176].log_data[0].max := 1.0, [1176].log_data[0].total := 300.0, [1176].log_data[0].time := 300.0, [1176].log_data[0].minminute := 30, [1176].log_data[0].maxminute := 30, [1176].log_data[0].valid := 1, [1176].log_data[1].valid := 1, [1176].log_data[2].valid := 1, [1176].log_data[3].valid := 1, [1176].log_data[4].valid := 1,
        [1176].time.Year := 2022, [1176].time.Month := 4, [1176].time.Day := 27, [1176].time.Hour := 23, [1176].time.Minute := 34, [1176].time.Second := 59, [1176].time.DST_ON := 1, [1177].log_data[0].min := 1.0, [1177].log_data[0].max := 1.0, [1177].log_data[0].total := 300.0, [1177].log_data[0].time := 300.0, [1177].log_data[0].minminute := 35, [1177].log_data[0].maxminute := 35, [1177].log_data[0].valid := 1, [1177].log_data[1].valid := 1, [1177].log_data[2].valid := 1, [1177].log_data[3].valid := 1, [1177].log_data[4].valid := 1, [1177].time.Year := 2022, [1177].time.Month := 4, [1177].time.Day := 27, [1177].time.Hour := 23, [1177].time.Minute := 39, [1177].time.Second := 59, [1177].time.DST_ON := 1, [1178].log_data[0].min := 1.0, [1178].log_data[0].max := 1.0, [1178].log_data[0].total := 300.0, [1178].log_data[0].time := 300.0, [1178].log_data[0].minminute := 40, [1178].log_data[0].maxminute := 40, [1178].log_data[0].valid := 1, [1178].log_data[1].valid := 1, [1178].log_data[2].valid := 1, [1178].log_data[3].valid := 1, [1178].log_data[4].valid := 1, [1178].time.Year := 2022, [1178].time.Month := 4, [1178].time.Day := 27, [1178].time.Hour := 23, [1178].time.Minute := 44, [1178].time.Second := 59, [1178].time.DST_ON := 1, [1179].log_data[0].min := 1.0, [1179].log_data[0].max := 1.0, [1179].log_data[0].total := 300.0, [1179].log_data[0].time := 300.0, [1179].log_data[0].minminute := 45, [1179].log_data[0].maxminute := 45, [1179].log_data[0].valid := 1, [1179].log_data[1].valid := 1, [1179].log_data[2].valid := 1, [1179].log_data[3].valid := 1, [1179].log_data[4].valid := 1, [1179].time.Year := 2022, [1179].time.Month := 4, [1179].time.Day := 27, [1179].time.Hour := 23, [1179].time.Minute := 49, [1179].time.Second := 59,
        [1179].time.DST_ON := 1, [1180].log_data[0].min := 1.0, [1180].log_data[0].max := 1.0, [1180].log_data[0].total := 300.0, [1180].log_data[0].time := 300.0, [1180].log_data[0].minminute := 50, [1180].log_data[0].maxminute := 50, [1180].log_data[0].valid := 1, [1180].log_data[1].valid := 1, [1180].log_data[2].valid := 1, [1180].log_data[3].valid := 1, [1180].log_data[4].valid := 1, [1180].time.Year := 2022, [1180].time.Month := 4, [1180].time.Day := 27, [1180].time.Hour := 23, [1180].time.Minute := 54, [1180].time.Second := 59, [1180].time.DST_ON := 1, [1181].log_data[0].min := 1.0, [1181].log_data[0].max := 1.0, [1181].log_data[0].total := 300.0, [1181].log_data[0].time := 300.0, [1181].log_data[0].minminute := 55, [1181].log_data[0].maxminute := 55, [1181].log_data[0].valid := 1, [1181].log_data[1].valid := 1, [1181].log_data[2].valid := 1, [1181].log_data[3].valid := 1, [1181].log_data[4].valid := 1, [1181].time.Year := 2022, [1181].time.Month := 4, [1181].time.Day := 27, [1181].time.Hour := 23, [1181].time.Minute := 59, [1181].time.Second := 59, [1181].time.DST_ON := 1, [1182].log_data[0].min := 1.0, [1182].log_data[0].max := 1.0, [1182].log_data[0].total := 300.0, [1182].log_data[0].time := 300.0, [1182].log_data[0].valid := 1, [1182].log_data[1].valid := 1, [1182].log_data[2].valid := 1, [1182].log_data[3].valid := 1, [1182].log_data[4].valid := 1, [1182].time.Year := 2022, [1182].time.Month := 4, [1182].time.Day := 28, [1182].time.Minute := 4, [1182].time.Second := 59, [1182].time.DST_ON := 1, [1183].log_data[0].min := 1.0, [1183].log_data[0].max := 1.0, [1183].log_data[0].total := 300.0, [1183].log_data[0].time := 300.0, [1183].log_data[0].minminute := 5, [1183].log_data[0].maxminute := 5, [1183].log_data[0].valid := 1, [1183].log_data[1].valid := 1,
        [1183].log_data[2].valid := 1, [1183].log_data[3].valid := 1, [1183].log_data[4].valid := 1, [1183].time.Year := 2022, [1183].time.Month := 4, [1183].time.Day := 28, [1183].time.Minute := 9, [1183].time.Second := 59, [1183].time.DST_ON := 1, [1184].log_data[0].min := 1.0, [1184].log_data[0].max := 1.0, [1184].log_data[0].total := 300.0, [1184].log_data[0].time := 300.0, [1184].log_data[0].minminute := 10, [1184].log_data[0].maxminute := 10, [1184].log_data[0].valid := 1, [1184].log_data[1].valid := 1, [1184].log_data[2].valid := 1, [1184].log_data[3].valid := 1, [1184].log_data[4].valid := 1, [1184].time.Year := 2022, [1184].time.Month := 4, [1184].time.Day := 28, [1184].time.Minute := 14, [1184].time.Second := 59, [1184].time.DST_ON := 1, [1185].log_data[0].min := 1.0, [1185].log_data[0].max := 1.0, [1185].log_data[0].total := 300.0, [1185].log_data[0].time := 300.0, [1185].log_data[0].minminute := 15, [1185].log_data[0].maxminute := 15, [1185].log_data[0].valid := 1, [1185].log_data[1].valid := 1, [1185].log_data[2].valid := 1, [1185].log_data[3].valid := 1, [1185].log_data[4].valid := 1, [1185].time.Year := 2022, [1185].time.Month := 4, [1185].time.Day := 28, [1185].time.Minute := 19, [1185].time.Second := 59, [1185].time.DST_ON := 1, [1186].log_data[0].min := 1.0, [1186].log_data[0].max := 1.0, [1186].log_data[0].total := 300.0, [1186].log_data[0].time := 300.0, [1186].log_data[0].minminute := 20, [1186].log_data[0].maxminute := 20, [1186].log_data[0].valid := 1, [1186].log_data[1].valid := 1, [1186].log_data[2].valid := 1, [1186].log_data[3].valid := 1, [1186].log_data[4].valid := 1, [1186].time.Year := 2022, [1186].time.Month := 4, [1186].time.Day := 28, [1186].time.Minute := 24, [1186].time.Second := 59, [1186].time.DST_ON := 1,
        [1187].log_data[0].min := 1.0, [1187].log_data[0].max := 1.0, [1187].log_data[0].total := 300.0, [1187].log_data[0].time := 300.0, [1187].log_data[0].minminute := 25, [1187].log_data[0].maxminute := 25, [1187].log_data[0].valid := 1, [1187].log_data[1].valid := 1, [1187].log_data[2].valid := 1, [1187].log_data[3].valid := 1, [1187].log_data[4].valid := 1, [1187].time.Year := 2022, [1187].time.Month := 4, [1187].time.Day := 28, [1187].time.Minute := 29, [1187].time.Second := 59, [1187].time.DST_ON := 1, [1188].log_data[0].min := 1.0, [1188].log_data[0].max := 1.0, [1188].log_data[0].total := 300.0, [1188].log_data[0].time := 300.0, [1188].log_data[0].minminute := 30, [1188].log_data[0].maxminute := 30, [1188].log_data[0].valid := 1, [1188].log_data[1].valid := 1, [1188].log_data[2].valid := 1, [1188].log_data[3].valid := 1, [1188].log_data[4].valid := 1, [1188].time.Year := 2022, [1188].time.Month := 4, [1188].time.Day := 28, [1188].time.Minute := 34, [1188].time.Second := 59, [1188].time.DST_ON := 1, [1189].log_data[0].min := 1.0, [1189].log_data[0].max := 1.0, [1189].log_data[0].total := 300.0, [1189].log_data[0].time := 300.0, [1189].log_data[0].minminute := 35, [1189].log_data[0].maxminute := 35, [1189].log_data[0].valid := 1, [1189].log_data[1].valid := 1, [1189].log_data[2].valid := 1, [1189].log_data[3].valid := 1, [1189].log_data[4].valid := 1, [1189].time.Year := 2022, [1189].time.Month := 4, [1189].time.Day := 28, [1189].time.Minute := 39, [1189].time.Second := 59, [1189].time.DST_ON := 1, [1190].log_data[0].min := 1.0, [1190].log_data[0].max := 1.0, [1190].log_data[0].total := 300.0, [1190].log_data[0].time := 300.0, [1190].log_data[0].minminute := 40, [1190].log_data[0].maxminute := 40, [1190].log_data[0].valid := 1, [1190].log_data[1].valid := 1, [1190].log_data[2].valid := 1,
        [1190].log_data[3].valid := 1, [1190].log_data[4].valid := 1, [1190].time.Year := 2022, [1190].time.Month := 4, [1190].time.Day := 28, [1190].time.Minute := 44, [1190].time.Second := 59, [1190].time.DST_ON := 1, [1191].log_data[0].min := 1.0, [1191].log_data[0].max := 1.0, [1191].log_data[0].total := 300.0, [1191].log_data[0].time := 300.0, [1191].log_data[0].minminute := 45, [1191].log_data[0].maxminute := 45, [1191].log_data[0].valid := 1, [1191].log_data[1].valid := 1, [1191].log_data[2].valid := 1, [1191].log_data[3].valid := 1, [1191].log_data[4].valid := 1, [1191].time.Year := 2022, [1191].time.Month := 4, [1191].time.Day := 28, [1191].time.Minute := 49, [1191].time.Second := 59, [1191].time.DST_ON := 1, [1192].log_data[0].min := 1.0, [1192].log_data[0].max := 1.0, [1192].log_data[0].total := 300.0, [1192].log_data[0].time := 300.0, [1192].log_data[0].minminute := 50, [1192].log_data[0].maxminute := 50, [1192].log_data[0].valid := 1, [1192].log_data[1].valid := 1, [1192].log_data[2].valid := 1, [1192].log_data[3].valid := 1, [1192].log_data[4].valid := 1, [1192].time.Year := 2022, [1192].time.Month := 4, [1192].time.Day := 28, [1192].time.Minute := 54, [1192].time.Second := 59, [1192].time.DST_ON := 1, [1193].log_data[0].min := 1.0, [1193].log_data[0].max := 1.0, [1193].log_data[0].total := 300.0, [1193].log_data[0].time := 300.0, [1193].log_data[0].minminute := 55, [1193].log_data[0].maxminute := 55, [1193].log_data[0].valid := 1, [1193].log_data[1].valid := 1, [1193].log_data[2].valid := 1, [1193].log_data[3].valid := 1, [1193].log_data[4].valid := 1, [1193].time.Year := 2022, [1193].time.Month := 4, [1193].time.Day := 28, [1193].time.Minute := 59, [1193].time.Second := 59, [1193].time.DST_ON := 1, [1194].log_data[0].min := 1.0,
        [1194].log_data[0].max := 1.0, [1194].log_data[0].total := 300.0, [1194].log_data[0].time := 300.0, [1194].log_data[0].valid := 1, [1194].log_data[1].valid := 1, [1194].log_data[2].valid := 1, [1194].log_data[3].valid := 1, [1194].log_data[4].valid := 1, [1194].time.Year := 2022, [1194].time.Month := 4, [1194].time.Day := 28, [1194].time.Hour := 1, [1194].time.Minute := 4, [1194].time.Second := 59, [1194].time.DST_ON := 1, [1195].log_data[0].min := 1.0, [1195].log_data[0].max := 1.0, [1195].log_data[0].total := 300.0, [1195].log_data[0].time := 300.0, [1195].log_data[0].minminute := 5, [1195].log_data[0].maxminute := 5, [1195].log_data[0].valid := 1, [1195].log_data[1].valid := 1, [1195].log_data[2].valid := 1, [1195].log_data[3].valid := 1, [1195].log_data[4].valid := 1, [1195].time.Year := 2022, [1195].time.Month := 4, [1195].time.Day := 28, [1195].time.Hour := 1, [1195].time.Minute := 9, [1195].time.Second := 59, [1195].time.DST_ON := 1, [1196].log_data[0].min := 1.0, [1196].log_data[0].max := 1.0, [1196].log_data[0].total := 300.0, [1196].log_data[0].time := 300.0, [1196].log_data[0].minminute := 10, [1196].log_data[0].maxminute := 10, [1196].log_data[0].valid := 1, [1196].log_data[1].valid := 1, [1196].log_data[2].valid := 1, [1196].log_data[3].valid := 1, [1196].log_data[4].valid := 1, [1196].time.Year := 2022, [1196].time.Month := 4, [1196].time.Day := 28, [1196].time.Hour := 1, [1196].time.Minute := 14, [1196].time.Second := 59, [1196].time.DST_ON := 1, [1197].log_data[0].min := 1.0, [1197].log_data[0].max := 1.0, [1197].log_data[0].total := 300.0, [1197].log_data[0].time := 300.0, [1197].log_data[0].minminute := 15, [1197].log_data[0].maxminute := 15, [1197].log_data[0].valid := 1, [1197].log_data[1].valid := 1, [1197].log_data[2].valid := 1,
        [1197].log_data[3].valid := 1, [1197].log_data[4].valid := 1, [1197].time.Year := 2022, [1197].time.Month := 4, [1197].time.Day := 28, [1197].time.Hour := 1, [1197].time.Minute := 19, [1197].time.Second := 59, [1197].time.DST_ON := 1, [1198].log_data[0].min := 1.0, [1198].log_data[0].max := 1.0, [1198].log_data[0].total := 300.0, [1198].log_data[0].time := 300.0, [1198].log_data[0].minminute := 20, [1198].log_data[0].maxminute := 20, [1198].log_data[0].valid := 1, [1198].log_data[1].valid := 1, [1198].log_data[2].valid := 1, [1198].log_data[3].valid := 1, [1198].log_data[4].valid := 1, [1198].time.Year := 2022, [1198].time.Month := 4, [1198].time.Day := 28, [1198].time.Hour := 1, [1198].time.Minute := 24, [1198].time.Second := 59, [1198].time.DST_ON := 1, [1199].log_data[0].min := 1.0, [1199].log_data[0].max := 1.0, [1199].log_data[0].total := 300.0, [1199].log_data[0].time := 300.0, [1199].log_data[0].minminute := 25, [1199].log_data[0].maxminute := 25, [1199].log_data[0].valid := 1, [1199].log_data[1].valid := 1, [1199].log_data[2].valid := 1, [1199].log_data[3].valid := 1, [1199].log_data[4].valid := 1, [1199].time.Year := 2022, [1199].time.Month := 4, [1199].time.Day := 28, [1199].time.Hour := 1, [1199].time.Minute := 29, [1199].time.Second := 59, [1199].time.DST_ON := 1, [1200].log_data[0].min := 1.0, [1200].log_data[0].max := 1.0, [1200].log_data[0].total := 300.0, [1200].log_data[0].time := 300.0, [1200].log_data[0].minminute := 30, [1200].log_data[0].maxminute := 30, [1200].log_data[0].valid := 1, [1200].log_data[1].valid := 1, [1200].log_data[2].valid := 1, [1200].log_data[3].valid := 1, [1200].log_data[4].valid := 1, [1200].time.Year := 2022, [1200].time.Month := 4, [1200].time.Day := 28, [1200].time.Hour := 1,
        [1200].time.Minute := 34, [1200].time.Second := 59, [1200].time.DST_ON := 1, [1201].log_data[0].min := 1.0, [1201].log_data[0].max := 1.0, [1201].log_data[0].total := 300.0, [1201].log_data[0].time := 300.0, [1201].log_data[0].minminute := 35, [1201].log_data[0].maxminute := 35, [1201].log_data[0].valid := 1, [1201].log_data[1].valid := 1, [1201].log_data[2].valid := 1, [1201].log_data[3].valid := 1, [1201].log_data[4].valid := 1, [1201].time.Year := 2022, [1201].time.Month := 4, [1201].time.Day := 28, [1201].time.Hour := 1, [1201].time.Minute := 39, [1201].time.Second := 59, [1201].time.DST_ON := 1, [1202].log_data[0].min := 1.0, [1202].log_data[0].max := 1.0, [1202].log_data[0].total := 300.0, [1202].log_data[0].time := 300.0, [1202].log_data[0].minminute := 40, [1202].log_data[0].maxminute := 40, [1202].log_data[0].valid := 1, [1202].log_data[1].valid := 1, [1202].log_data[2].valid := 1, [1202].log_data[3].valid := 1, [1202].log_data[4].valid := 1, [1202].time.Year := 2022, [1202].time.Month := 4, [1202].time.Day := 28, [1202].time.Hour := 1, [1202].time.Minute := 44, [1202].time.Second := 59, [1202].time.DST_ON := 1, [1203].log_data[0].min := 1.0, [1203].log_data[0].max := 1.0, [1203].log_data[0].total := 300.0, [1203].log_data[0].time := 300.0, [1203].log_data[0].minminute := 45, [1203].log_data[0].maxminute := 45, [1203].log_data[0].valid := 1, [1203].log_data[1].valid := 1, [1203].log_data[2].valid := 1, [1203].log_data[3].valid := 1, [1203].log_data[4].valid := 1, [1203].time.Year := 2022, [1203].time.Month := 4, [1203].time.Day := 28, [1203].time.Hour := 1, [1203].time.Minute := 49, [1203].time.Second := 59, [1203].time.DST_ON := 1, [1204].log_data[0].min := 1.0, [1204].log_data[0].max := 1.0, [1204].log_data[0].total := 300.0,
        [1204].log_data[0].time := 300.0, [1204].log_data[0].minminute := 50, [1204].log_data[0].maxminute := 50, [1204].log_data[0].valid := 1, [1204].log_data[1].valid := 1, [1204].log_data[2].valid := 1, [1204].log_data[3].valid := 1, [1204].log_data[4].valid := 1, [1204].time.Year := 2022, [1204].time.Month := 4, [1204].time.Day := 28, [1204].time.Hour := 1, [1204].time.Minute := 54, [1204].time.Second := 59, [1204].time.DST_ON := 1, [1205].log_data[0].min := 1.0, [1205].log_data[0].max := 1.0, [1205].log_data[0].total := 300.0, [1205].log_data[0].time := 300.0, [1205].log_data[0].minminute := 55, [1205].log_data[0].maxminute := 55, [1205].log_data[0].valid := 1, [1205].log_data[1].valid := 1, [1205].log_data[2].valid := 1, [1205].log_data[3].valid := 1, [1205].log_data[4].valid := 1, [1205].time.Year := 2022, [1205].time.Month := 4, [1205].time.Day := 28, [1205].time.Hour := 1, [1205].time.Minute := 59, [1205].time.Second := 59, [1205].time.DST_ON := 1, [1206].log_data[0].min := 1.0, [1206].log_data[0].max := 1.0, [1206].log_data[0].total := 300.0, [1206].log_data[0].time := 300.0, [1206].log_data[0].valid := 1, [1206].log_data[1].valid := 1, [1206].log_data[2].valid := 1, [1206].log_data[3].valid := 1, [1206].log_data[4].valid := 1, [1206].time.Year := 2022, [1206].time.Month := 4, [1206].time.Day := 28, [1206].time.Hour := 2, [1206].time.Minute := 4, [1206].time.Second := 59, [1206].time.DST_ON := 1, [1207].log_data[0].min := 1.0, [1207].log_data[0].max := 1.0, [1207].log_data[0].total := 300.0, [1207].log_data[0].time := 300.0, [1207].log_data[0].minminute := 5, [1207].log_data[0].maxminute := 5, [1207].log_data[0].valid := 1, [1207].log_data[1].valid := 1, [1207].log_data[2].valid := 1, [1207].log_data[3].valid := 1, [1207].log_data[4].valid := 1,
        [1207].time.Year := 2022, [1207].time.Month := 4, [1207].time.Day := 28, [1207].time.Hour := 2, [1207].time.Minute := 9, [1207].time.Second := 59, [1207].time.DST_ON := 1, [1208].log_data[0].min := 1.0, [1208].log_data[0].max := 1.0, [1208].log_data[0].total := 300.0, [1208].log_data[0].time := 300.0, [1208].log_data[0].minminute := 10, [1208].log_data[0].maxminute := 10, [1208].log_data[0].valid := 1, [1208].log_data[1].valid := 1, [1208].log_data[2].valid := 1, [1208].log_data[3].valid := 1, [1208].log_data[4].valid := 1, [1208].time.Year := 2022, [1208].time.Month := 4, [1208].time.Day := 28, [1208].time.Hour := 2, [1208].time.Minute := 14, [1208].time.Second := 59, [1208].time.DST_ON := 1, [1209].log_data[0].min := 1.0, [1209].log_data[0].max := 1.0, [1209].log_data[0].total := 300.0, [1209].log_data[0].time := 300.0, [1209].log_data[0].minminute := 15, [1209].log_data[0].maxminute := 15, [1209].log_data[0].valid := 1, [1209].log_data[1].valid := 1, [1209].log_data[2].valid := 1, [1209].log_data[3].valid := 1, [1209].log_data[4].valid := 1, [1209].time.Year := 2022, [1209].time.Month := 4, [1209].time.Day := 28, [1209].time.Hour := 2, [1209].time.Minute := 19, [1209].time.Second := 59, [1209].time.DST_ON := 1, [1210].log_data[0].min := 1.0, [1210].log_data[0].max := 1.0, [1210].log_data[0].total := 300.0, [1210].log_data[0].time := 300.0, [1210].log_data[0].minminute := 20, [1210].log_data[0].maxminute := 20, [1210].log_data[0].valid := 1, [1210].log_data[1].valid := 1, [1210].log_data[2].valid := 1, [1210].log_data[3].valid := 1, [1210].log_data[4].valid := 1, [1210].time.Year := 2022, [1210].time.Month := 4, [1210].time.Day := 28, [1210].time.Hour := 2, [1210].time.Minute := 24, [1210].time.Second := 59,
        [1210].time.DST_ON := 1, [1211].log_data[0].min := 1.0, [1211].log_data[0].max := 1.0, [1211].log_data[0].total := 300.0, [1211].log_data[0].time := 300.0, [1211].log_data[0].minminute := 25, [1211].log_data[0].maxminute := 25, [1211].log_data[0].valid := 1, [1211].log_data[1].valid := 1, [1211].log_data[2].valid := 1, [1211].log_data[3].valid := 1, [1211].log_data[4].valid := 1, [1211].time.Year := 2022, [1211].time.Month := 4, [1211].time.Day := 28, [1211].time.Hour := 2, [1211].time.Minute := 29, [1211].time.Second := 59, [1211].time.DST_ON := 1, [1212].log_data[0].min := 1.0, [1212].log_data[0].max := 1.0, [1212].log_data[0].total := 300.0, [1212].log_data[0].time := 300.0, [1212].log_data[0].minminute := 30, [1212].log_data[0].maxminute := 30, [1212].log_data[0].valid := 1, [1212].log_data[1].valid := 1, [1212].log_data[2].valid := 1, [1212].log_data[3].valid := 1, [1212].log_data[4].valid := 1, [1212].time.Year := 2022, [1212].time.Month := 4, [1212].time.Day := 28, [1212].time.Hour := 2, [1212].time.Minute := 34, [1212].time.Second := 59, [1212].time.DST_ON := 1, [1213].log_data[0].min := 1.0, [1213].log_data[0].max := 1.0, [1213].log_data[0].total := 300.0, [1213].log_data[0].time := 300.0, [1213].log_data[0].minminute := 35, [1213].log_data[0].maxminute := 35, [1213].log_data[0].valid := 1, [1213].log_data[1].valid := 1, [1213].log_data[2].valid := 1, [1213].log_data[3].valid := 1, [1213].log_data[4].valid := 1, [1213].time.Year := 2022, [1213].time.Month := 4, [1213].time.Day := 28, [1213].time.Hour := 2, [1213].time.Minute := 39, [1213].time.Second := 59, [1213].time.DST_ON := 1, [1214].log_data[0].min := 1.0, [1214].log_data[0].max := 1.0, [1214].log_data[0].total := 300.0, [1214].log_data[0].time := 300.0, [1214].log_data[0].minminute := 40,
        [1214].log_data[0].maxminute := 40, [1214].log_data[0].valid := 1, [1214].log_data[1].valid := 1, [1214].log_data[2].valid := 1, [1214].log_data[3].valid := 1, [1214].log_data[4].valid := 1, [1214].time.Year := 2022, [1214].time.Month := 4, [1214].time.Day := 28, [1214].time.Hour := 2, [1214].time.Minute := 44, [1214].time.Second := 59, [1214].time.DST_ON := 1, [1215].log_data[0].min := 1.0, [1215].log_data[0].max := 1.0, [1215].log_data[0].total := 300.0, [1215].log_data[0].time := 300.0, [1215].log_data[0].minminute := 45, [1215].log_data[0].maxminute := 45, [1215].log_data[0].valid := 1, [1215].log_data[1].valid := 1, [1215].log_data[2].valid := 1, [1215].log_data[3].valid := 1, [1215].log_data[4].valid := 1, [1215].time.Year := 2022, [1215].time.Month := 4, [1215].time.Day := 28, [1215].time.Hour := 2, [1215].time.Minute := 49, [1215].time.Second := 59, [1215].time.DST_ON := 1, [1216].log_data[0].min := 1.0, [1216].log_data[0].max := 1.0, [1216].log_data[0].total := 300.0, [1216].log_data[0].time := 300.0, [1216].log_data[0].minminute := 50, [1216].log_data[0].maxminute := 50, [1216].log_data[0].valid := 1, [1216].log_data[1].valid := 1, [1216].log_data[2].valid := 1, [1216].log_data[3].valid := 1, [1216].log_data[4].valid := 1, [1216].time.Year := 2022, [1216].time.Month := 4, [1216].time.Day := 28, [1216].time.Hour := 2, [1216].time.Minute := 54, [1216].time.Second := 59, [1216].time.DST_ON := 1, [1217].log_data[0].min := 1.0, [1217].log_data[0].max := 1.0, [1217].log_data[0].total := 300.0, [1217].log_data[0].time := 300.0, [1217].log_data[0].minminute := 55, [1217].log_data[0].maxminute := 55, [1217].log_data[0].valid := 1, [1217].log_data[1].valid := 1, [1217].log_data[2].valid := 1, [1217].log_data[3].valid := 1, [1217].log_data[4].valid := 1,
        [1217].time.Year := 2022, [1217].time.Month := 4, [1217].time.Day := 28, [1217].time.Hour := 2, [1217].time.Minute := 59, [1217].time.Second := 59, [1217].time.DST_ON := 1, [1218].log_data[0].min := 1.0, [1218].log_data[0].max := 1.0, [1218].log_data[0].total := 300.0, [1218].log_data[0].time := 300.0, [1218].log_data[0].valid := 1, [1218].log_data[1].valid := 1, [1218].log_data[2].valid := 1, [1218].log_data[3].valid := 1, [1218].log_data[4].valid := 1, [1218].time.Year := 2022, [1218].time.Month := 4, [1218].time.Day := 28, [1218].time.Hour := 3, [1218].time.Minute := 4, [1218].time.Second := 59, [1218].time.DST_ON := 1, [1219].log_data[0].min := 1.0, [1219].log_data[0].max := 1.0, [1219].log_data[0].total := 300.0, [1219].log_data[0].time := 300.0, [1219].log_data[0].minminute := 5, [1219].log_data[0].maxminute := 5, [1219].log_data[0].valid := 1, [1219].log_data[1].valid := 1, [1219].log_data[2].valid := 1, [1219].log_data[3].valid := 1, [1219].log_data[4].valid := 1, [1219].time.Year := 2022, [1219].time.Month := 4, [1219].time.Day := 28, [1219].time.Hour := 3, [1219].time.Minute := 9, [1219].time.Second := 59, [1219].time.DST_ON := 1, [1220].log_data[0].min := 1.0, [1220].log_data[0].max := 1.0, [1220].log_data[0].total := 300.0, [1220].log_data[0].time := 300.0, [1220].log_data[0].minminute := 10, [1220].log_data[0].maxminute := 10, [1220].log_data[0].valid := 1, [1220].log_data[1].valid := 1, [1220].log_data[2].valid := 1, [1220].log_data[3].valid := 1, [1220].log_data[4].valid := 1, [1220].time.Year := 2022, [1220].time.Month := 4, [1220].time.Day := 28, [1220].time.Hour := 3, [1220].time.Minute := 14, [1220].time.Second := 59, [1220].time.DST_ON := 1, [1221].log_data[0].min := 1.0,
        [1221].log_data[0].max := 1.0, [1221].log_data[0].total := 300.0, [1221].log_data[0].time := 300.0, [1221].log_data[0].minminute := 15, [1221].log_data[0].maxminute := 15, [1221].log_data[0].valid := 1, [1221].log_data[1].valid := 1, [1221].log_data[2].valid := 1, [1221].log_data[3].valid := 1, [1221].log_data[4].valid := 1, [1221].time.Year := 2022, [1221].time.Month := 4, [1221].time.Day := 28, [1221].time.Hour := 3, [1221].time.Minute := 19, [1221].time.Second := 59, [1221].time.DST_ON := 1, [1222].log_data[0].min := 1.0, [1222].log_data[0].max := 1.0, [1222].log_data[0].total := 300.0, [1222].log_data[0].time := 300.0, [1222].log_data[0].minminute := 20, [1222].log_data[0].maxminute := 20, [1222].log_data[0].valid := 1, [1222].log_data[1].valid := 1, [1222].log_data[2].valid := 1, [1222].log_data[3].valid := 1, [1222].log_data[4].valid := 1, [1222].time.Year := 2022, [1222].time.Month := 4, [1222].time.Day := 28, [1222].time.Hour := 3, [1222].time.Minute := 24, [1222].time.Second := 59, [1222].time.DST_ON := 1, [1223].log_data[0].min := 1.0, [1223].log_data[0].max := 1.0, [1223].log_data[0].total := 300.0, [1223].log_data[0].time := 300.0, [1223].log_data[0].minminute := 25, [1223].log_data[0].maxminute := 25, [1223].log_data[0].valid := 1, [1223].log_data[1].valid := 1, [1223].log_data[2].valid := 1, [1223].log_data[3].valid := 1, [1223].log_data[4].valid := 1, [1223].time.Year := 2022, [1223].time.Month := 4, [1223].time.Day := 28, [1223].time.Hour := 3, [1223].time.Minute := 29, [1223].time.Second := 59, [1223].time.DST_ON := 1, [1224].log_data[0].min := 1.0, [1224].log_data[0].max := 1.0, [1224].log_data[0].total := 300.0, [1224].log_data[0].time := 300.0, [1224].log_data[0].minminute := 30, [1224].log_data[0].maxminute := 30, [1224].log_data[0].valid := 1,
        [1224].log_data[1].valid := 1, [1224].log_data[2].valid := 1, [1224].log_data[3].valid := 1, [1224].log_data[4].valid := 1, [1224].time.Year := 2022, [1224].time.Month := 4, [1224].time.Day := 28, [1224].time.Hour := 3, [1224].time.Minute := 34, [1224].time.Second := 59, [1224].time.DST_ON := 1, [1225].log_data[0].min := 1.0, [1225].log_data[0].max := 1.0, [1225].log_data[0].total := 300.0, [1225].log_data[0].time := 300.0, [1225].log_data[0].minminute := 35, [1225].log_data[0].maxminute := 35, [1225].log_data[0].valid := 1, [1225].log_data[1].valid := 1, [1225].log_data[2].valid := 1, [1225].log_data[3].valid := 1, [1225].log_data[4].valid := 1, [1225].time.Year := 2022, [1225].time.Month := 4, [1225].time.Day := 28, [1225].time.Hour := 3, [1225].time.Minute := 39, [1225].time.Second := 59, [1225].time.DST_ON := 1, [1226].log_data[0].min := 1.0, [1226].log_data[0].max := 1.0, [1226].log_data[0].total := 299.999, [1226].log_data[0].time := 299.999, [1226].log_data[0].minminute := 40, [1226].log_data[0].maxminute := 40, [1226].log_data[0].valid := 1, [1226].log_data[1].valid := 1, [1226].log_data[2].valid := 1, [1226].log_data[3].valid := 1, [1226].log_data[4].valid := 1, [1226].time.Year := 2022, [1226].time.Month := 4, [1226].time.Day := 28, [1226].time.Hour := 3, [1226].time.Minute := 44, [1226].time.Second := 59, [1226].time.DST_ON := 1, [1227].log_data[0].min := 1.0, [1227].log_data[0].max := 1.0, [1227].log_data[0].total := 300.0, [1227].log_data[0].time := 300.0, [1227].log_data[0].minminute := 45, [1227].log_data[0].maxminute := 45, [1227].log_data[0].valid := 1, [1227].log_data[1].valid := 1, [1227].log_data[2].valid := 1, [1227].log_data[3].valid := 1, [1227].log_data[4].valid := 1, [1227].time.Year := 2022, [1227].time.Month := 4,
        [1227].time.Day := 28, [1227].time.Hour := 3, [1227].time.Minute := 49, [1227].time.Second := 59, [1227].time.DST_ON := 1, [1228].log_data[0].min := 1.0, [1228].log_data[0].max := 1.0, [1228].log_data[0].total := 300.0, [1228].log_data[0].time := 300.0, [1228].log_data[0].minminute := 50, [1228].log_data[0].maxminute := 50, [1228].log_data[0].valid := 1, [1228].log_data[1].valid := 1, [1228].log_data[2].valid := 1, [1228].log_data[3].valid := 1, [1228].log_data[4].valid := 1, [1228].time.Year := 2022, [1228].time.Month := 4, [1228].time.Day := 28, [1228].time.Hour := 3, [1228].time.Minute := 54, [1228].time.Second := 59, [1228].time.DST_ON := 1, [1229].log_data[0].min := 1.0, [1229].log_data[0].max := 1.0, [1229].log_data[0].total := 300.0, [1229].log_data[0].time := 300.0, [1229].log_data[0].minminute := 55, [1229].log_data[0].maxminute := 55, [1229].log_data[0].valid := 1, [1229].log_data[1].valid := 1, [1229].log_data[2].valid := 1, [1229].log_data[3].valid := 1, [1229].log_data[4].valid := 1, [1229].time.Year := 2022, [1229].time.Month := 4, [1229].time.Day := 28, [1229].time.Hour := 3, [1229].time.Minute := 59, [1229].time.Second := 59, [1229].time.DST_ON := 1, [1230].log_data[0].min := 1.0, [1230].log_data[0].max := 1.0, [1230].log_data[0].total := 300.0, [1230].log_data[0].time := 300.0, [1230].log_data[0].valid := 1, [1230].log_data[1].valid := 1, [1230].log_data[2].valid := 1, [1230].log_data[3].valid := 1, [1230].log_data[4].valid := 1, [1230].time.Year := 2022, [1230].time.Month := 4, [1230].time.Day := 28, [1230].time.Hour := 4, [1230].time.Minute := 4, [1230].time.Second := 59, [1230].time.DST_ON := 1, [1231].log_data[0].min := 1.0, [1231].log_data[0].max := 1.0, [1231].log_data[0].total := 300.0,
        [1231].log_data[0].time := 300.0, [1231].log_data[0].minminute := 5, [1231].log_data[0].maxminute := 5, [1231].log_data[0].valid := 1, [1231].log_data[1].valid := 1, [1231].log_data[2].valid := 1, [1231].log_data[3].valid := 1, [1231].log_data[4].valid := 1, [1231].time.Year := 2022, [1231].time.Month := 4, [1231].time.Day := 28, [1231].time.Hour := 4, [1231].time.Minute := 9, [1231].time.Second := 59, [1231].time.DST_ON := 1, [1232].log_data[0].min := 1.0, [1232].log_data[0].max := 1.0, [1232].log_data[0].total := 300.0, [1232].log_data[0].time := 300.0, [1232].log_data[0].minminute := 10, [1232].log_data[0].maxminute := 10, [1232].log_data[0].valid := 1, [1232].log_data[1].valid := 1, [1232].log_data[2].valid := 1, [1232].log_data[3].valid := 1, [1232].log_data[4].valid := 1, [1232].time.Year := 2022, [1232].time.Month := 4, [1232].time.Day := 28, [1232].time.Hour := 4, [1232].time.Minute := 14, [1232].time.Second := 59, [1232].time.DST_ON := 1, [1233].log_data[0].min := 1.0, [1233].log_data[0].max := 1.0, [1233].log_data[0].total := 300.0, [1233].log_data[0].time := 300.0, [1233].log_data[0].minminute := 15, [1233].log_data[0].maxminute := 15, [1233].log_data[0].valid := 1, [1233].log_data[1].valid := 1, [1233].log_data[2].valid := 1, [1233].log_data[3].valid := 1, [1233].log_data[4].valid := 1, [1233].time.Year := 2022, [1233].time.Month := 4, [1233].time.Day := 28, [1233].time.Hour := 4, [1233].time.Minute := 19, [1233].time.Second := 59, [1233].time.DST_ON := 1, [1234].log_data[0].min := 1.0, [1234].log_data[0].max := 1.0, [1234].log_data[0].total := 300.0, [1234].log_data[0].time := 300.0, [1234].log_data[0].minminute := 20, [1234].log_data[0].maxminute := 20, [1234].log_data[0].valid := 1, [1234].log_data[1].valid := 1, [1234].log_data[2].valid := 1,
        [1234].log_data[3].valid := 1, [1234].log_data[4].valid := 1, [1234].time.Year := 2022, [1234].time.Month := 4, [1234].time.Day := 28, [1234].time.Hour := 4, [1234].time.Minute := 24, [1234].time.Second := 59, [1234].time.DST_ON := 1, [1235].log_data[0].min := 1.0, [1235].log_data[0].max := 1.0, [1235].log_data[0].total := 300.0, [1235].log_data[0].time := 300.0, [1235].log_data[0].minminute := 25, [1235].log_data[0].maxminute := 25, [1235].log_data[0].valid := 1, [1235].log_data[1].valid := 1, [1235].log_data[2].valid := 1, [1235].log_data[3].valid := 1, [1235].log_data[4].valid := 1, [1235].time.Year := 2022, [1235].time.Month := 4, [1235].time.Day := 28, [1235].time.Hour := 4, [1235].time.Minute := 29, [1235].time.Second := 59, [1235].time.DST_ON := 1, [1236].log_data[0].min := 1.0, [1236].log_data[0].max := 1.0, [1236].log_data[0].total := 300.0, [1236].log_data[0].time := 300.0, [1236].log_data[0].minminute := 30, [1236].log_data[0].maxminute := 30, [1236].log_data[0].valid := 1, [1236].log_data[1].valid := 1, [1236].log_data[2].valid := 1, [1236].log_data[3].valid := 1, [1236].log_data[4].valid := 1, [1236].time.Year := 2022, [1236].time.Month := 4, [1236].time.Day := 28, [1236].time.Hour := 4, [1236].time.Minute := 34, [1236].time.Second := 59, [1236].time.DST_ON := 1, [1237].log_data[0].min := 1.0, [1237].log_data[0].max := 1.0, [1237].log_data[0].total := 300.0, [1237].log_data[0].time := 300.0, [1237].log_data[0].minminute := 35, [1237].log_data[0].maxminute := 35, [1237].log_data[0].valid := 1, [1237].log_data[1].valid := 1, [1237].log_data[2].valid := 1, [1237].log_data[3].valid := 1, [1237].log_data[4].valid := 1, [1237].time.Year := 2022, [1237].time.Month := 4, [1237].time.Day := 28, [1237].time.Hour := 4,
        [1237].time.Minute := 39, [1237].time.Second := 59, [1237].time.DST_ON := 1, [1238].log_data[0].min := 1.0, [1238].log_data[0].max := 1.0, [1238].log_data[0].total := 300.0, [1238].log_data[0].time := 300.0, [1238].log_data[0].minminute := 40, [1238].log_data[0].maxminute := 40, [1238].log_data[0].valid := 1, [1238].log_data[1].valid := 1, [1238].log_data[2].valid := 1, [1238].log_data[3].valid := 1, [1238].log_data[4].valid := 1, [1238].time.Year := 2022, [1238].time.Month := 4, [1238].time.Day := 28, [1238].time.Hour := 4, [1238].time.Minute := 44, [1238].time.Second := 59, [1238].time.DST_ON := 1, [1239].log_data[0].min := 1.0, [1239].log_data[0].max := 1.0, [1239].log_data[0].total := 300.0, [1239].log_data[0].time := 300.0, [1239].log_data[0].minminute := 45, [1239].log_data[0].maxminute := 45, [1239].log_data[0].valid := 1, [1239].log_data[1].valid := 1, [1239].log_data[2].valid := 1, [1239].log_data[3].valid := 1, [1239].log_data[4].valid := 1, [1239].time.Year := 2022, [1239].time.Month := 4, [1239].time.Day := 28, [1239].time.Hour := 4, [1239].time.Minute := 49, [1239].time.Second := 59, [1239].time.DST_ON := 1, [1240].log_data[0].min := 1.0, [1240].log_data[0].max := 1.0, [1240].log_data[0].total := 300.0, [1240].log_data[0].time := 300.0, [1240].log_data[0].minminute := 50, [1240].log_data[0].maxminute := 50, [1240].log_data[0].valid := 1, [1240].log_data[1].valid := 1, [1240].log_data[2].valid := 1, [1240].log_data[3].valid := 1, [1240].log_data[4].valid := 1, [1240].time.Year := 2022, [1240].time.Month := 4, [1240].time.Day := 28, [1240].time.Hour := 4, [1240].time.Minute := 54, [1240].time.Second := 59, [1240].time.DST_ON := 1, [1241].log_data[0].min := 1.0, [1241].log_data[0].max := 1.0, [1241].log_data[0].total := 300.0,
